KUKA KRL program: PPR-mid-01.src

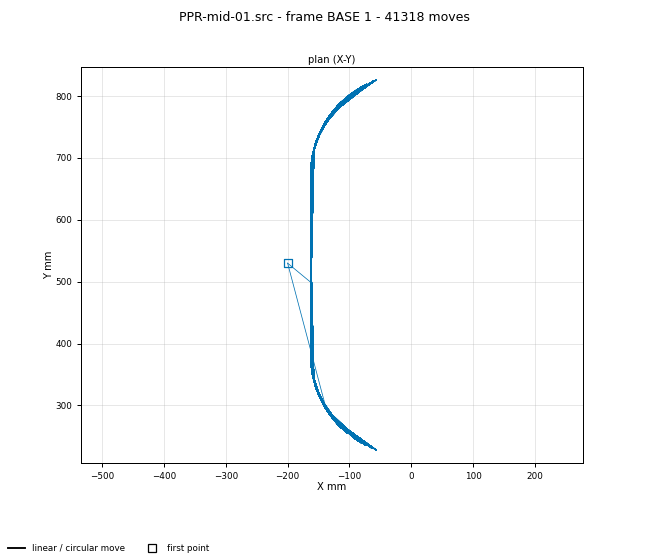
[picture p0: tool path of PPR-mid-01.src in frame BASE 1, 41318 of 41319 moves have a stored position in this frame; points joined in program order, loops and branches not executed]
&ACCESS RVEO
&REL 11
&PARAM TEMPLATE = C:\KRC\Roboter\Template\vorgabe
&PARAM EDITMASK = *
DEF variable_helical2( )
;FOLD INI
  ;FOLD BASISTECH INI
    GLOBAL INTERRUPT DECL 3 WHEN $STOPMESS==TRUE DO IR_STOPM ( )
    INTERRUPT ON 3
    BAS (#INITMOV,0 )
  ;ENDFOLD (BASISTECH INI)
 ;FOLD USER INI


    ;Make your modifications here
  ;ENDFOLD (USER INI)
;ENDFOLD (INI)
ACTION(#AXIS_RESET,34,1000,#NOERROR,ERROR_CODE)
;FOLD PTP HOME  Vel= 100 % DEFAULT;%{PE}%MKUKATPBASIS,%CMOVE,%VPTP,%P 1:PTP, 2:HOME, 3:, 5:100, 7:DEFAULT
$BWDSTART = FALSE
PDAT_ACT=PDEFAULT
FDAT_ACT=FHOME
BAS (#PTP_PARAMS,100 )
$H_POS=XHOME
PTP  XHOME
;ENDFOLD
BAS(#TOOL,1)
BAS(#BASE,1)
$VEL_AXIS[1]=100
$VEL_AXIS[2]=100
$VEL_AXIS[3]=100
$VEL_AXIS[4]=100
$VEL_AXIS[5]=100
$VEL_AXIS[6]=100
$VEL_EXTAX[1]=100
$VEL_EXTAX[2]=100

$ACC_AXIS[1]=100
$ACC_AXIS[2]=100
$ACC_AXIS[3]=100
$ACC_AXIS[4]=100
$ACC_AXIS[5]=100
$ACC_AXIS[6]=100
$ACC_EXTAX[1]=100
$ACC_EXTAX[2]=100

;;;;;;;;; postprocessing parameters (date 2024-01-25T18:14:56.965272)
; qxconst: -162.82
; qxconstarcys: -149.5,143.5
; qE3offset: 0.00
; qyoffset: 530.00
; qswitchsplit: 3
; qthinningtol: 0.2010
;;;;;;;;;

SLIN {X  -200.000, Y  +530.000, Z    +0.000, A    +0.000, E1    +0.000, E3    +0.000, E4    +0.000}

SLIN {X  -137.186, Y  +292.805, Z    +0.000, E1   +73.993, E3   +38.340}
HALT
SPLINE
SPL {X  -133.270, Y  +286.961, Z    +0.000, E1   +73.739, E3   +43.054}
SPL {X  -130.283, Y  +282.844, Z    +0.000, E1   +73.297, E3   +47.946}
SPL {X  -126.880, Y  +278.461, Z    +0.000, E1   +72.855, E3   +52.696}
SPL {X  -123.363, Y  +274.237, Z    +0.000, E1   +72.376, E3   +57.178}
SPL {X  -121.018, Y  +271.573, Z    +0.000, E1   +72.049, E3   +59.863}
SPL {X  -113.980, Y  +264.229, Z    +0.000, E1   +74.120, E3   +55.442}
SPL {X   -56.216, Y  +227.692, Z    +0.000, E1   +56.267, E3  +232.166}
ENDSPLINE

SPLINE
SPL {X  -126.995, Y  +278.604, Z    +0.000, E1   +59.937, E3  +404.406}
SPL {X  -150.196, Y  +317.640, Z    +0.000, E1   +49.956, E3  +412.861}
SPL {X  -157.261, Y  +338.316, Z    +0.000, E1   +40.017, E3  +414.556}
SPL {X  -160.924, Y  +355.726, Z    +0.000, E1   +27.715, E3  +414.997}
SPL {X  -162.423, Y  +369.141, Z    +0.000, E1   +15.207, E3  +415.432}
SPL {X  -162.811, Y  +378.755, Z    +0.000, E1    +4.616, E3  +415.347}
SPL {X  -162.820, Y  +382.684, Z    +0.000, E1    -0.227, E3  +414.902}
SPL {X  -162.820, Y  +385.721, Z    +0.000, E1    -8.371, E3  +414.717}
SPL {X  -162.820, Y  +388.532, Z    +0.000, E1   -16.412, E3  +414.604}
SPL {X  -162.820, Y  +392.558, Z    +0.000, E1   -27.778, E3  +414.692}
SPL {X  -162.820, Y  +400.474, Z    +0.000, E1   -46.251, E3  +414.556}
SPL {X  -162.820, Y  +414.510, Z    +0.000, E1   -65.115, E3  +413.999}
SPL {X  -162.820, Y  +465.064, Z    +0.000, E1   -76.269, E3  +423.847}
SPL {X  -157.184, Y  +715.968, Z    +0.000, E1   -76.600, E3  +519.805}
SPL {X  -156.461, Y  +718.560, Z    +0.000, E1   -75.553, E3  +533.225}
SPL {X  -151.911, Y  +732.096, Z    +0.000, E1   -75.235, E3  +543.779}
SPL {X  -146.569, Y  +744.407, Z    +0.000, E1   -74.677, E3  +555.583}
SPL {X  -142.375, Y  +752.491, Z    +0.000, E1   -74.335, E3  +562.610}
SPL {X  -139.539, Y  +757.399, Z    +0.000, E1   -73.892, E3  +568.808}
SPL {X  -136.017, Y  +762.997, Z    +0.000, E1   -73.579, E3  +573.990}
SPL {X  -133.089, Y  +767.296, Z    +0.000, E1   -73.251, E3  +578.448}
SPL {X  -129.985, Y  +771.553, Z    +0.000, E1   -72.801, E3  +583.442}
SPL {X  -126.581, Y  +775.909, Z    +0.000, E1   -72.426, E3  +587.753}
SPL {X  -122.528, Y  +780.725, Z    +0.000, E1   -71.905, E3  +592.773}
SPL {X  -116.189, Y  +787.563, Z    +0.000, E1   -72.978, E3  +592.058}
SPL {X   -57.587, Y  +825.796, Z    +0.000, E1   -56.753, E3  +747.309}
ENDSPLINE

SPLINE
SPL {X  -124.075, Y  +778.932, Z    +0.000, E1   -61.393, E3  +940.938}
SPL {X  -150.653, Y  +735.257, Z    +0.000, E1   -50.160, E3  +948.618}
SPL {X  -159.377, Y  +706.804, Z    +0.000, E1   -34.828, E3  +950.261}
SPL {X  -162.134, Y  +688.425, Z    +0.000, E1   -19.100, E3  +950.198}
SPL {X  -162.734, Y  +678.779, Z    +0.000, E1    -8.745, E3  +950.337}
SPL {X  -162.820, Y  +671.589, Z    +0.000, E1    -0.221, E3  +949.971}
SPL {X  -162.820, Y  +669.743, Z    +0.000, E1    +4.352, E3  +949.746}
SPL {X  -162.820, Y  +665.917, Z    +0.000, E1   +15.272, E3  +949.740}
SPL {X  -162.820, Y  +661.245, Z    +0.000, E1   +28.879, E3  +949.581}
SPL {X  -162.820, Y  +654.015, Z    +0.000, E1   +45.814, E3  +949.728}
SPL {X  -162.820, Y  +641.345, Z    +0.000, E1   +63.138, E3  +949.775}
SPL {X  -162.820, Y  +620.039, Z    +0.000, E1   +75.979, E3  +948.385}
SPL {X  -162.820, Y  +571.094, Z    +0.000, E1   +77.089, E3  +963.564}
SPL {X  -157.487, Y  +339.169, Z    +0.000, E1   +76.425, E3 +1056.668}
SPL {X  -156.386, Y  +335.181, Z    +0.000, E1   +75.555, E3 +1068.729}
SPL {X  -152.710, Y  +324.020, Z    +0.000, E1   +75.365, E3 +1076.539}
SPL {X  -139.497, Y  +296.529, Z    +0.000, E1   +77.231, E3 +1070.111}
ENDSPLINE

SPLINE
SPL {X  -139.792, Y  +297.022, Z    +0.000, E1   +76.273, E3 +1078.806}
ENDSPLINE

SPLINE
SPL {X  -138.933, Y  +295.600, Z    +0.000, E1   +75.173, E3 +1089.289}
SPL {X  -137.186, Y  +292.805, Z    +0.000, E1   +73.993, E3 +1099.879}
SPL {X  -133.270, Y  +286.961, Z    +0.000, E1   +73.739, E3 +1104.592}
SPL {X  -130.283, Y  +282.844, Z    +0.000, E1   +73.297, E3 +1109.484}
SPL {X  -127.795, Y  +279.610, Z    +0.000, E1   +72.860, E3 +1113.614}
SPL {X  -124.650, Y  +275.749, Z    +0.000, E1   +72.674, E3 +1116.533}
SPL {X  -121.687, Y  +272.322, Z    +0.000, E1   +72.100, E3 +1120.842}
SPL {X  -113.980, Y  +264.229, Z    +0.000, E1   +74.120, E3 +1116.980}
SPL {X   -56.216, Y  +227.692, Z    +0.000, E1   +56.267, E3 +1293.704}
ENDSPLINE

SPLINE
SPL {X  -126.995, Y  +278.604, Z    +0.000, E1   +59.937, E3 +1465.945}
SPL {X  -150.196, Y  +317.640, Z    +0.000, E1   +49.956, E3 +1474.400}
SPL {X  -157.261, Y  +338.316, Z    +0.000, E1   +40.017, E3 +1476.095}
SPL {X  -160.924, Y  +355.726, Z    +0.000, E1   +27.715, E3 +1476.535}
SPL {X  -162.423, Y  +369.141, Z    +0.000, E1   +15.207, E3 +1476.971}
SPL {X  -162.811, Y  +378.755, Z    +0.000, E1    +4.616, E3 +1476.885}
SPL {X  -162.820, Y  +382.684, Z    +0.000, E1    -0.227, E3 +1476.440}
SPL {X  -162.820, Y  +385.721, Z    +0.000, E1    -8.371, E3 +1476.256}
SPL {X  -162.820, Y  +388.532, Z    +0.000, E1   -16.412, E3 +1476.142}
SPL {X  -162.820, Y  +392.558, Z    +0.000, E1   -27.778, E3 +1476.231}
SPL {X  -162.820, Y  +398.468, Z    +0.000, E1   -42.446, E3 +1476.081}
SPL {X  -162.820, Y  +404.415, Z    +0.000, E1   -53.236, E3 +1476.121}
SPL {X  -162.820, Y  +414.510, Z    +0.000, E1   -65.115, E3 +1475.538}
SPL {X  -162.820, Y  +457.766, Z    +0.000, E1   -75.929, E3 +1483.374}
SPL {X  -162.820, Y  +471.144, Z    +0.000, E1   -76.496, E3 +1487.063}
SPL {X  -158.097, Y  +712.432, Z    +0.000, E1   -77.677, E3 +1567.773}
SPL {X  -156.557, Y  +718.224, Z    +0.000, E1   -75.715, E3 +1592.910}
SPL {X  -153.015, Y  +729.150, Z    +0.000, E1   -75.312, E3 +1602.852}
SPL {X  -149.053, Y  +739.025, Z    +0.000, E1   -74.952, E3 +1611.648}
SPL {X  -144.053, Y  +749.389, Z    +0.000, E1   -74.457, E3 +1621.639}
SPL {X  -139.539, Y  +757.399, Z    +0.000, E1   -73.892, E3 +1630.346}
SPL {X  -136.017, Y  +762.997, Z    +0.000, E1   -73.579, E3 +1635.529}
SPL {X  -133.089, Y  +767.296, Z    +0.000, E1   -73.251, E3 +1639.987}
SPL {X  -129.985, Y  +771.553, Z    +0.000, E1   -72.801, E3 +1644.981}
SPL {X  -126.581, Y  +775.909, Z    +0.000, E1   -72.426, E3 +1649.292}
SPL {X  -123.329, Y  +779.803, Z    +0.000, E1   -71.936, E3 +1653.674}
SPL {X  -119.291, Y  +784.315, Z    +0.000, E1   -72.148, E3 +1655.085}
SPL {X   -57.587, Y  +825.796, Z    +0.000, E1   -56.753, E3 +1808.848}
ENDSPLINE

SPLINE
SPL {X  -124.075, Y  +778.932, Z    +0.000, E1   -61.393, E3 +2002.477}
SPL {X  -150.653, Y  +735.257, Z    +0.000, E1   -50.160, E3 +2010.156}
SPL {X  -159.377, Y  +706.804, Z    +0.000, E1   -34.828, E3 +2011.800}
SPL {X  -162.134, Y  +688.425, Z    +0.000, E1   -19.100, E3 +2011.736}
SPL {X  -162.803, Y  +675.871, Z    +0.000, E1    -5.469, E3 +2011.920}
SPL {X  -162.820, Y  +671.500, Z    +0.000, E1    +0.000, E3 +2011.488}
SPL {X  -162.820, Y  +669.743, Z    +0.000, E1    +4.352, E3 +2011.284}
SPL {X  -162.820, Y  +665.917, Z    +0.000, E1   +15.272, E3 +2011.279}
SPL {X  -162.820, Y  +661.245, Z    +0.000, E1   +28.879, E3 +2011.120}
SPL {X  -162.820, Y  +654.015, Z    +0.000, E1   +45.814, E3 +2011.267}
SPL {X  -162.820, Y  +641.345, Z    +0.000, E1   +63.138, E3 +2011.314}
SPL {X  -162.820, Y  +620.039, Z    +0.000, E1   +75.979, E3 +2009.924}
SPL {X  -162.820, Y  +571.094, Z    +0.000, E1   +77.089, E3 +2025.102}
SPL {X  -157.487, Y  +339.169, Z    +0.000, E1   +76.425, E3 +2118.206}
SPL {X  -156.386, Y  +335.181, Z    +0.000, E1   +75.555, E3 +2130.267}
SPL {X  -152.710, Y  +324.020, Z    +0.000, E1   +75.365, E3 +2138.077}
SPL {X  -139.497, Y  +296.529, Z    +0.000, E1   +77.231, E3 +2131.649}
ENDSPLINE

SPLINE
SPL {X  -139.792, Y  +297.022, Z    +0.000, E1   +76.273, E3 +2140.344}
ENDSPLINE

SPLINE
SPL {X  -138.933, Y  +295.600, Z    +0.000, E1   +75.173, E3 +2150.827}
SPL {X  -137.186, Y  +292.805, Z    +0.000, E1   +73.993, E3 +2161.417}
SPL {X  -133.270, Y  +286.961, Z    +0.000, E1   +73.739, E3 +2166.131}
SPL {X  -130.283, Y  +282.844, Z    +0.000, E1   +73.297, E3 +2171.023}
SPL {X  -127.795, Y  +279.610, Z    +0.000, E1   +72.860, E3 +2175.153}
SPL {X  -124.650, Y  +275.749, Z    +0.000, E1   +72.674, E3 +2178.071}
SPL {X  -121.687, Y  +272.322, Z    +0.000, E1   +72.100, E3 +2182.381}
SPL {X  -113.980, Y  +264.229, Z    +0.000, E1   +74.120, E3 +2178.519}
SPL {X   -56.216, Y  +227.692, Z    +0.000, E1   +56.267, E3 +2355.243}
ENDSPLINE

SPLINE
SPL {X  -126.995, Y  +278.604, Z    +0.000, E1   +59.937, E3 +2527.483}
SPL {X  -150.196, Y  +317.640, Z    +0.000, E1   +49.956, E3 +2535.938}
SPL {X  -157.261, Y  +338.316, Z    +0.000, E1   +40.017, E3 +2537.633}
SPL {X  -160.924, Y  +355.726, Z    +0.000, E1   +27.715, E3 +2538.074}
SPL {X  -162.423, Y  +369.141, Z    +0.000, E1   +15.207, E3 +2538.509}
SPL {X  -162.811, Y  +378.755, Z    +0.000, E1    +4.616, E3 +2538.424}
SPL {X  -162.820, Y  +382.684, Z    +0.000, E1    -0.227, E3 +2537.978}
SPL {X  -162.820, Y  +387.227, Z    +0.000, E1   -12.320, E3 +2537.733}
SPL {X  -162.820, Y  +392.558, Z    +0.000, E1   -27.778, E3 +2537.769}
SPL {X  -162.820, Y  +400.474, Z    +0.000, E1   -46.251, E3 +2537.633}
SPL {X  -162.820, Y  +414.510, Z    +0.000, E1   -65.115, E3 +2537.076}
SPL {X  -162.820, Y  +465.064, Z    +0.000, E1   -76.269, E3 +2546.924}
SPL {X  -158.097, Y  +712.432, Z    +0.000, E1   -77.677, E3 +2629.312}
SPL {X  -156.557, Y  +718.224, Z    +0.000, E1   -75.715, E3 +2654.448}
SPL {X  -151.911, Y  +732.096, Z    +0.000, E1   -75.235, E3 +2666.856}
SPL {X  -146.569, Y  +744.407, Z    +0.000, E1   -74.677, E3 +2678.660}
SPL {X  -142.375, Y  +752.491, Z    +0.000, E1   -74.335, E3 +2685.687}
SPL {X  -139.539, Y  +757.399, Z    +0.000, E1   -73.892, E3 +2691.885}
SPL {X  -136.017, Y  +762.997, Z    +0.000, E1   -73.579, E3 +2697.067}
SPL {X  -133.089, Y  +767.296, Z    +0.000, E1   -73.251, E3 +2701.525}
SPL {X  -129.985, Y  +771.553, Z    +0.000, E1   -72.801, E3 +2706.519}
SPL {X  -126.581, Y  +775.909, Z    +0.000, E1   -72.426, E3 +2710.830}
SPL {X  -123.329, Y  +779.803, Z    +0.000, E1   -71.936, E3 +2715.212}
SPL {X  -119.291, Y  +784.315, Z    +0.000, E1   -72.148, E3 +2716.624}
SPL {X   -57.587, Y  +825.796, Z    +0.000, E1   -56.753, E3 +2870.386}
ENDSPLINE

SPLINE
SPL {X  -124.075, Y  +778.932, Z    +0.000, E1   -61.393, E3 +3064.015}
SPL {X  -150.653, Y  +735.257, Z    +0.000, E1   -50.160, E3 +3071.695}
SPL {X  -159.377, Y  +706.804, Z    +0.000, E1   -34.828, E3 +3073.338}
SPL {X  -162.134, Y  +688.425, Z    +0.000, E1   -19.100, E3 +3073.275}
SPL {X  -162.803, Y  +675.871, Z    +0.000, E1    -5.469, E3 +3073.459}
SPL {X  -162.820, Y  +671.500, Z    +0.000, E1    +0.000, E3 +3073.027}
SPL {X  -162.820, Y  +669.743, Z    +0.000, E1    +4.352, E3 +3072.822}
SPL {X  -162.820, Y  +665.917, Z    +0.000, E1   +15.272, E3 +3072.817}
SPL {X  -162.820, Y  +661.245, Z    +0.000, E1   +28.879, E3 +3072.658}
SPL {X  -162.820, Y  +654.015, Z    +0.000, E1   +45.814, E3 +3072.805}
SPL {X  -162.820, Y  +641.345, Z    +0.000, E1   +63.138, E3 +3072.852}
SPL {X  -162.820, Y  +620.039, Z    +0.000, E1   +75.979, E3 +3071.462}
SPL {X  -162.820, Y  +571.094, Z    +0.000, E1   +77.089, E3 +3086.641}
SPL {X  -157.487, Y  +339.169, Z    +0.000, E1   +76.425, E3 +3179.745}
SPL {X  -156.386, Y  +335.181, Z    +0.000, E1   +75.555, E3 +3191.805}
SPL {X  -152.710, Y  +324.020, Z    +0.000, E1   +75.365, E3 +3199.616}
SPL {X  -139.497, Y  +296.529, Z    +0.000, E1   +77.231, E3 +3193.188}
ENDSPLINE

SPLINE
SPL {X  -139.792, Y  +297.022, Z    +0.000, E1   +76.273, E3 +3201.883}
ENDSPLINE

SPLINE
SPL {X  -138.933, Y  +295.600, Z    +0.000, E1   +75.173, E3 +3212.365}
SPL {X  -137.186, Y  +292.805, Z    +0.000, E1   +73.993, E3 +3222.956}
SPL {X  -133.270, Y  +286.961, Z    +0.000, E1   +73.739, E3 +3227.669}
SPL {X  -130.283, Y  +282.844, Z    +0.000, E1   +73.297, E3 +3232.561}
SPL {X  -127.795, Y  +279.610, Z    +0.000, E1   +72.860, E3 +3236.691}
SPL {X  -124.650, Y  +275.749, Z    +0.000, E1   +72.674, E3 +3239.610}
SPL {X  -121.687, Y  +272.322, Z    +0.000, E1   +72.100, E3 +3243.919}
SPL {X  -113.980, Y  +264.229, Z    +0.000, E1   +74.120, E3 +3240.057}
SPL {X   -56.216, Y  +227.692, Z    +0.000, E1   +56.267, E3 +3416.781}
ENDSPLINE

SPLINE
SPL {X  -126.995, Y  +278.604, Z    +0.000, E1   +59.937, E3 +3589.021}
SPL {X  -150.196, Y  +317.640, Z    +0.000, E1   +49.956, E3 +3597.477}
SPL {X  -157.261, Y  +338.316, Z    +0.000, E1   +40.017, E3 +3599.172}
SPL {X  -160.924, Y  +355.726, Z    +0.000, E1   +27.715, E3 +3599.612}
SPL {X  -162.423, Y  +369.141, Z    +0.000, E1   +15.207, E3 +3600.048}
SPL {X  -162.811, Y  +378.755, Z    +0.000, E1    +4.616, E3 +3599.962}
SPL {X  -162.820, Y  +382.684, Z    +0.000, E1    -0.227, E3 +3599.517}
SPL {X  -162.820, Y  +387.227, Z    +0.000, E1   -12.320, E3 +3599.272}
SPL {X  -162.820, Y  +392.558, Z    +0.000, E1   -27.778, E3 +3599.308}
SPL {X  -162.820, Y  +400.474, Z    +0.000, E1   -46.251, E3 +3599.172}
SPL {X  -162.820, Y  +414.510, Z    +0.000, E1   -65.115, E3 +3598.615}
SPL {X  -162.820, Y  +465.064, Z    +0.000, E1   -76.269, E3 +3608.463}
SPL {X  -158.097, Y  +712.432, Z    +0.000, E1   -77.677, E3 +3690.850}
SPL {X  -156.557, Y  +718.224, Z    +0.000, E1   -75.715, E3 +3715.987}
SPL {X  -151.911, Y  +732.096, Z    +0.000, E1   -75.235, E3 +3728.394}
SPL {X  -146.569, Y  +744.407, Z    +0.000, E1   -74.677, E3 +3740.198}
SPL {X  -142.375, Y  +752.491, Z    +0.000, E1   -74.335, E3 +3747.226}
SPL {X  -139.539, Y  +757.399, Z    +0.000, E1   -73.892, E3 +3753.423}
SPL {X  -136.017, Y  +762.997, Z    +0.000, E1   -73.579, E3 +3758.606}
SPL {X  -133.089, Y  +767.296, Z    +0.000, E1   -73.251, E3 +3763.064}
SPL {X  -129.985, Y  +771.553, Z    +0.000, E1   -72.801, E3 +3768.057}
SPL {X  -126.581, Y  +775.909, Z    +0.000, E1   -72.426, E3 +3772.369}
SPL {X  -123.329, Y  +779.803, Z    +0.000, E1   -71.936, E3 +3776.750}
SPL {X  -119.291, Y  +784.315, Z    +0.000, E1   -72.148, E3 +3778.162}
SPL {X   -57.587, Y  +825.796, Z    +0.000, E1   -56.753, E3 +3931.925}
ENDSPLINE

SPLINE
SPL {X  -124.075, Y  +778.932, Z    +0.000, E1   -61.393, E3 +4125.554}
SPL {X  -150.653, Y  +735.257, Z    +0.000, E1   -50.160, E3 +4133.233}
SPL {X  -159.377, Y  +706.804, Z    +0.000, E1   -34.828, E3 +4134.876}
SPL {X  -162.134, Y  +688.425, Z    +0.000, E1   -19.100, E3 +4134.813}
SPL {X  -162.803, Y  +675.871, Z    +0.000, E1    -5.469, E3 +4134.997}
SPL {X  -162.820, Y  +671.500, Z    +0.000, E1    +0.000, E3 +4134.565}
SPL {X  -162.820, Y  +669.743, Z    +0.000, E1    +4.352, E3 +4134.361}
SPL {X  -162.820, Y  +665.917, Z    +0.000, E1   +15.272, E3 +4134.355}
SPL {X  -162.820, Y  +661.245, Z    +0.000, E1   +28.879, E3 +4134.197}
SPL {X  -162.820, Y  +654.015, Z    +0.000, E1   +45.814, E3 +4134.344}
SPL {X  -162.820, Y  +641.345, Z    +0.000, E1   +63.138, E3 +4134.391}
SPL {X  -162.820, Y  +620.039, Z    +0.000, E1   +75.979, E3 +4133.001}
SPL {X  -162.820, Y  +571.094, Z    +0.000, E1   +77.089, E3 +4148.179}
SPL {X  -157.487, Y  +339.169, Z    +0.000, E1   +76.425, E3 +4241.283}
SPL {X  -156.386, Y  +335.181, Z    +0.000, E1   +75.555, E3 +4253.344}
SPL {X  -152.710, Y  +324.020, Z    +0.000, E1   +75.365, E3 +4261.154}
SPL {X  -139.497, Y  +296.529, Z    +0.000, E1   +77.231, E3 +4254.726}
ENDSPLINE

SPLINE
SPL {X  -139.792, Y  +297.022, Z    +0.000, E1   +76.273, E3 +4263.421}
ENDSPLINE

SPLINE
SPL {X  -138.933, Y  +295.600, Z    +0.000, E1   +75.173, E3 +4273.904}
SPL {X  -137.186, Y  +292.805, Z    +0.000, E1   +73.993, E3 +4284.494}
SPL {X  -133.270, Y  +286.961, Z    +0.000, E1   +73.739, E3 +4289.208}
SPL {X  -130.283, Y  +282.844, Z    +0.000, E1   +73.297, E3 +4294.100}
SPL {X  -127.795, Y  +279.610, Z    +0.000, E1   +72.860, E3 +4298.230}
SPL {X  -124.650, Y  +275.749, Z    +0.000, E1   +72.674, E3 +4301.148}
SPL {X  -121.687, Y  +272.322, Z    +0.000, E1   +72.100, E3 +4305.457}
SPL {X  -113.980, Y  +264.229, Z    +0.000, E1   +74.120, E3 +4301.596}
SPL {X   -56.216, Y  +227.692, Z    +0.000, E1   +56.267, E3 +4478.320}
ENDSPLINE

SPLINE
SPL {X  -126.995, Y  +278.604, Z    +0.000, E1   +59.937, E3 +4650.560}
SPL {X  -150.196, Y  +317.640, Z    +0.000, E1   +49.956, E3 +4659.015}
SPL {X  -157.261, Y  +338.316, Z    +0.000, E1   +40.017, E3 +4660.710}
SPL {X  -160.924, Y  +355.726, Z    +0.000, E1   +27.715, E3 +4661.151}
SPL {X  -162.423, Y  +369.141, Z    +0.000, E1   +15.207, E3 +4661.586}
SPL {X  -162.811, Y  +378.755, Z    +0.000, E1    +4.616, E3 +4661.501}
SPL {X  -162.820, Y  +382.684, Z    +0.000, E1    -0.227, E3 +4661.055}
SPL {X  -162.820, Y  +387.227, Z    +0.000, E1   -12.320, E3 +4660.810}
SPL {X  -162.820, Y  +392.558, Z    +0.000, E1   -27.778, E3 +4660.846}
SPL {X  -162.820, Y  +400.474, Z    +0.000, E1   -46.251, E3 +4660.710}
SPL {X  -162.820, Y  +414.510, Z    +0.000, E1   -65.115, E3 +4660.153}
SPL {X  -162.820, Y  +465.064, Z    +0.000, E1   -76.269, E3 +4670.001}
SPL {X  -158.097, Y  +712.432, Z    +0.000, E1   -77.677, E3 +4752.389}
SPL {X  -156.557, Y  +718.224, Z    +0.000, E1   -75.715, E3 +4777.525}
SPL {X  -151.911, Y  +732.096, Z    +0.000, E1   -75.235, E3 +4789.932}
SPL {X  -146.569, Y  +744.407, Z    +0.000, E1   -74.677, E3 +4801.737}
SPL {X  -142.375, Y  +752.491, Z    +0.000, E1   -74.335, E3 +4808.764}
SPL {X  -139.539, Y  +757.399, Z    +0.000, E1   -73.892, E3 +4814.962}
SPL {X  -136.017, Y  +762.997, Z    +0.000, E1   -73.579, E3 +4820.144}
SPL {X  -133.089, Y  +767.296, Z    +0.000, E1   -73.251, E3 +4824.602}
SPL {X  -129.985, Y  +771.553, Z    +0.000, E1   -72.801, E3 +4829.596}
SPL {X  -126.581, Y  +775.909, Z    +0.000, E1   -72.426, E3 +4833.907}
SPL {X  -123.329, Y  +779.803, Z    +0.000, E1   -71.936, E3 +4838.289}
SPL {X  -119.291, Y  +784.315, Z    +0.000, E1   -72.148, E3 +4839.701}
SPL {X   -57.587, Y  +825.796, Z    +0.000, E1   -56.753, E3 +4993.463}
ENDSPLINE

SPLINE
SPL {X  -124.075, Y  +778.932, Z    +0.000, E1   -61.393, E3 +5187.092}
SPL {X  -150.653, Y  +735.257, Z    +0.000, E1   -50.160, E3 +5194.772}
SPL {X  -159.377, Y  +706.804, Z    +0.000, E1   -34.828, E3 +5196.415}
SPL {X  -162.134, Y  +688.425, Z    +0.000, E1   -19.100, E3 +5196.352}
SPL {X  -162.803, Y  +675.871, Z    +0.000, E1    -5.469, E3 +5196.536}
SPL {X  -162.820, Y  +671.500, Z    +0.000, E1    +0.000, E3 +5196.104}
SPL {X  -162.820, Y  +669.743, Z    +0.000, E1    +4.352, E3 +5195.899}
SPL {X  -162.820, Y  +665.917, Z    +0.000, E1   +15.272, E3 +5195.894}
SPL {X  -162.820, Y  +661.245, Z    +0.000, E1   +28.879, E3 +5195.735}
SPL {X  -162.820, Y  +654.015, Z    +0.000, E1   +45.814, E3 +5195.882}
SPL {X  -162.820, Y  +641.345, Z    +0.000, E1   +63.138, E3 +5195.929}
SPL {X  -162.820, Y  +620.039, Z    +0.000, E1   +75.979, E3 +5194.539}
SPL {X  -162.820, Y  +571.094, Z    +0.000, E1   +77.089, E3 +5209.718}
SPL {X  -157.487, Y  +339.169, Z    +0.000, E1   +76.425, E3 +5302.822}
SPL {X  -156.386, Y  +335.181, Z    +0.000, E1   +75.555, E3 +5314.882}
SPL {X  -152.710, Y  +324.020, Z    +0.000, E1   +75.365, E3 +5322.693}
SPL {X  -139.497, Y  +296.529, Z    +0.000, E1   +77.231, E3 +5316.264}
ENDSPLINE

SPLINE
SPL {X  -139.520, Y  +296.568, Z    +0.000, E1   +75.884, E3 +5328.912}
ENDSPLINE

SPLINE
SPL {X  -138.554, Y  +294.984, Z    +0.000, E1   +74.772, E3 +5338.793}
SPL {X  -137.186, Y  +292.805, Z    +0.000, E1   +73.993, E3 +5346.033}
SPL {X  -133.270, Y  +286.961, Z    +0.000, E1   +73.739, E3 +5350.746}
SPL {X  -130.283, Y  +282.844, Z    +0.000, E1   +73.297, E3 +5355.638}
SPL {X  -126.880, Y  +278.461, Z    +0.000, E1   +72.855, E3 +5360.389}
SPL {X  -123.363, Y  +274.237, Z    +0.000, E1   +72.376, E3 +5364.871}
SPL {X  -121.018, Y  +271.573, Z    +0.000, E1   +72.049, E3 +5367.556}
SPL {X  -113.980, Y  +264.229, Z    +0.000, E1   +74.120, E3 +5363.134}
SPL {X   -56.216, Y  +227.692, Z    +0.000, E1   +56.267, E3 +5539.858}
ENDSPLINE

SPLINE
SPL {X  -126.995, Y  +278.604, Z    +0.000, E1   +59.937, E3 +5712.098}
SPL {X  -150.196, Y  +317.640, Z    +0.000, E1   +49.956, E3 +5720.553}
SPL {X  -157.261, Y  +338.316, Z    +0.000, E1   +40.017, E3 +5722.249}
SPL {X  -160.924, Y  +355.726, Z    +0.000, E1   +27.715, E3 +5722.689}
SPL {X  -162.423, Y  +369.141, Z    +0.000, E1   +15.207, E3 +5723.125}
SPL {X  -162.811, Y  +378.755, Z    +0.000, E1    +4.616, E3 +5723.039}
SPL {X  -162.820, Y  +382.684, Z    +0.000, E1    -0.227, E3 +5722.594}
SPL {X  -162.820, Y  +385.721, Z    +0.000, E1    -8.371, E3 +5722.409}
SPL {X  -162.820, Y  +388.532, Z    +0.000, E1   -16.412, E3 +5722.296}
SPL {X  -162.820, Y  +392.558, Z    +0.000, E1   -27.778, E3 +5722.385}
SPL {X  -162.820, Y  +400.474, Z    +0.000, E1   -46.251, E3 +5722.248}
SPL {X  -162.820, Y  +414.510, Z    +0.000, E1   -65.115, E3 +5721.692}
SPL {X  -162.820, Y  +465.064, Z    +0.000, E1   -76.269, E3 +5731.540}
SPL {X  -157.184, Y  +715.968, Z    +0.000, E1   -76.600, E3 +5827.497}
SPL {X  -156.461, Y  +718.560, Z    +0.000, E1   -75.553, E3 +5840.917}
SPL {X  -153.015, Y  +729.150, Z    +0.000, E1   -75.312, E3 +5849.006}
SPL {X  -149.053, Y  +739.025, Z    +0.000, E1   -74.952, E3 +5857.802}
SPL {X  -144.053, Y  +749.389, Z    +0.000, E1   -74.457, E3 +5867.793}
SPL {X  -139.539, Y  +757.399, Z    +0.000, E1   -73.892, E3 +5876.500}
SPL {X  -136.017, Y  +762.997, Z    +0.000, E1   -73.579, E3 +5881.683}
SPL {X  -133.089, Y  +767.296, Z    +0.000, E1   -73.251, E3 +5886.141}
SPL {X  -129.985, Y  +771.553, Z    +0.000, E1   -72.801, E3 +5891.134}
SPL {X  -126.581, Y  +775.909, Z    +0.000, E1   -72.426, E3 +5895.446}
SPL {X  -123.329, Y  +779.803, Z    +0.000, E1   -71.936, E3 +5899.827}
SPL {X  -119.291, Y  +784.315, Z    +0.000, E1   -72.148, E3 +5901.239}
SPL {X   -57.587, Y  +825.796, Z    +0.000, E1   -56.753, E3 +6055.002}
ENDSPLINE

SPLINE
SPL {X  -124.075, Y  +778.932, Z    +0.000, E1   -61.393, E3 +6248.631}
SPL {X  -147.028, Y  +743.450, Z    +0.000, E1   -53.078, E3 +6255.368}
SPL {X  -152.552, Y  +730.406, Z    +0.000, E1   -48.136, E3 +6256.786}
SPL {X  -159.377, Y  +706.804, Z    +0.000, E1   -34.828, E3 +6257.953}
SPL {X  -162.134, Y  +688.425, Z    +0.000, E1   -19.100, E3 +6257.890}
SPL {X  -162.803, Y  +675.871, Z    +0.000, E1    -5.469, E3 +6258.074}
SPL {X  -162.820, Y  +671.500, Z    +0.000, E1    +0.000, E3 +6257.642}
SPL {X  -162.820, Y  +669.743, Z    +0.000, E1    +4.352, E3 +6257.438}
SPL {X  -162.820, Y  +665.917, Z    +0.000, E1   +15.272, E3 +6257.432}
SPL {X  -162.820, Y  +659.880, Z    +0.000, E1   +32.256, E3 +6257.344}
SPL {X  -162.820, Y  +652.069, Z    +0.000, E1   +49.663, E3 +6257.369}
SPL {X  -162.820, Y  +641.345, Z    +0.000, E1   +63.138, E3 +6257.468}
SPL {X  -162.820, Y  +620.039, Z    +0.000, E1   +75.979, E3 +6256.078}
SPL {X  -162.820, Y  +578.479, Z    +0.000, E1   +77.260, E3 +6268.348}
SPL {X  -162.820, Y  +557.052, Z    +0.000, E1   +76.772, E3 +6276.829}
SPL {X  -157.487, Y  +339.169, Z    +0.000, E1   +76.425, E3 +6364.360}
SPL {X  -156.386, Y  +335.181, Z    +0.000, E1   +75.555, E3 +6376.421}
SPL {X  -152.710, Y  +324.020, Z    +0.000, E1   +75.365, E3 +6384.231}
SPL {X  -139.497, Y  +296.529, Z    +0.000, E1   +77.231, E3 +6377.803}
ENDSPLINE

SPLINE
SPL {X  -139.520, Y  +296.568, Z    +0.000, E1   +75.884, E3 +6390.450}
ENDSPLINE

SPLINE
SPL {X  -138.554, Y  +294.984, Z    +0.000, E1   +74.772, E3 +6400.331}
SPL {X  -137.186, Y  +292.805, Z    +0.000, E1   +73.993, E3 +6407.571}
SPL {X  -133.270, Y  +286.961, Z    +0.000, E1   +73.739, E3 +6412.285}
SPL {X  -130.283, Y  +282.844, Z    +0.000, E1   +73.297, E3 +6417.177}
SPL {X  -126.880, Y  +278.461, Z    +0.000, E1   +72.855, E3 +6421.927}
SPL {X  -123.363, Y  +274.237, Z    +0.000, E1   +72.376, E3 +6426.409}
SPL {X  -121.018, Y  +271.573, Z    +0.000, E1   +72.049, E3 +6429.094}
SPL {X  -113.980, Y  +264.229, Z    +0.000, E1   +74.120, E3 +6424.673}
SPL {X   -56.216, Y  +227.692, Z    +0.000, E1   +56.267, E3 +6601.397}
ENDSPLINE

SPLINE
SPL {X  -126.995, Y  +278.604, Z    +0.000, E1   +59.937, E3 +6773.637}
SPL {X  -150.196, Y  +317.640, Z    +0.000, E1   +49.956, E3 +6782.092}
SPL {X  -157.261, Y  +338.316, Z    +0.000, E1   +40.017, E3 +6783.787}
SPL {X  -160.924, Y  +355.726, Z    +0.000, E1   +27.715, E3 +6784.228}
SPL {X  -162.423, Y  +369.141, Z    +0.000, E1   +15.207, E3 +6784.663}
SPL {X  -162.811, Y  +378.755, Z    +0.000, E1    +4.616, E3 +6784.578}
SPL {X  -162.820, Y  +382.684, Z    +0.000, E1    -0.227, E3 +6784.132}
SPL {X  -162.820, Y  +385.721, Z    +0.000, E1    -8.371, E3 +6783.948}
SPL {X  -162.820, Y  +388.532, Z    +0.000, E1   -16.412, E3 +6783.834}
SPL {X  -162.820, Y  +392.558, Z    +0.000, E1   -27.778, E3 +6783.923}
SPL {X  -162.820, Y  +398.468, Z    +0.000, E1   -42.446, E3 +6783.774}
SPL {X  -162.820, Y  +404.415, Z    +0.000, E1   -53.236, E3 +6783.813}
SPL {X  -162.820, Y  +414.510, Z    +0.000, E1   -65.115, E3 +6783.230}
SPL {X  -162.820, Y  +457.766, Z    +0.000, E1   -75.929, E3 +6791.066}
SPL {X  -162.820, Y  +471.144, Z    +0.000, E1   -76.496, E3 +6794.755}
SPL {X  -158.097, Y  +712.432, Z    +0.000, E1   -77.677, E3 +6875.466}
SPL {X  -156.557, Y  +718.224, Z    +0.000, E1   -75.715, E3 +6900.602}
SPL {X  -151.911, Y  +732.096, Z    +0.000, E1   -75.235, E3 +6913.009}
SPL {X  -146.569, Y  +744.407, Z    +0.000, E1   -74.677, E3 +6924.814}
SPL {X  -142.375, Y  +752.491, Z    +0.000, E1   -74.335, E3 +6931.841}
SPL {X  -139.539, Y  +757.399, Z    +0.000, E1   -73.892, E3 +6938.039}
SPL {X  -136.017, Y  +762.997, Z    +0.000, E1   -73.579, E3 +6943.221}
SPL {X  -133.089, Y  +767.296, Z    +0.000, E1   -73.251, E3 +6947.679}
SPL {X  -129.985, Y  +771.553, Z    +0.000, E1   -72.801, E3 +6952.673}
SPL {X  -126.581, Y  +775.909, Z    +0.000, E1   -72.426, E3 +6956.984}
SPL {X  -123.329, Y  +779.803, Z    +0.000, E1   -71.936, E3 +6961.366}
SPL {X  -119.291, Y  +784.315, Z    +0.000, E1   -72.148, E3 +6962.778}
SPL {X   -57.587, Y  +825.796, Z    +0.000, E1   -56.753, E3 +7116.540}
ENDSPLINE

SPLINE
SPL {X  -124.075, Y  +778.932, Z    +0.000, E1   -61.393, E3 +7310.169}
SPL {X  -150.653, Y  +735.257, Z    +0.000, E1   -50.160, E3 +7317.848}
SPL {X  -159.377, Y  +706.804, Z    +0.000, E1   -34.828, E3 +7319.492}
SPL {X  -162.134, Y  +688.425, Z    +0.000, E1   -19.100, E3 +7319.429}
SPL {X  -162.734, Y  +678.779, Z    +0.000, E1    -8.745, E3 +7319.568}
SPL {X  -162.820, Y  +671.589, Z    +0.000, E1    -0.221, E3 +7319.202}
SPL {X  -162.820, Y  +669.743, Z    +0.000, E1    +4.352, E3 +7318.976}
SPL {X  -162.820, Y  +665.917, Z    +0.000, E1   +15.272, E3 +7318.971}
SPL {X  -162.820, Y  +659.880, Z    +0.000, E1   +32.256, E3 +7318.882}
SPL {X  -162.820, Y  +652.069, Z    +0.000, E1   +49.663, E3 +7318.908}
SPL {X  -162.820, Y  +641.345, Z    +0.000, E1   +63.138, E3 +7319.006}
SPL {X  -162.820, Y  +620.039, Z    +0.000, E1   +75.979, E3 +7317.616}
SPL {X  -162.820, Y  +571.094, Z    +0.000, E1   +77.089, E3 +7332.795}
SPL {X  -158.110, Y  +341.619, Z    +0.000, E1   +77.339, E3 +7414.444}
SPL {X  -156.597, Y  +335.917, Z    +0.000, E1   +75.680, E3 +7436.288}
SPL {X  -152.710, Y  +324.020, Z    +0.000, E1   +75.365, E3 +7445.770}
SPL {X  -139.497, Y  +296.529, Z    +0.000, E1   +77.231, E3 +7439.341}
ENDSPLINE

SPLINE
SPL {X  -139.792, Y  +297.022, Z    +0.000, E1   +76.273, E3 +7448.037}
ENDSPLINE

SPLINE
SPL {X  -138.933, Y  +295.600, Z    +0.000, E1   +75.173, E3 +7458.519}
SPL {X  -137.186, Y  +292.805, Z    +0.000, E1   +73.993, E3 +7469.110}
SPL {X  -133.270, Y  +286.961, Z    +0.000, E1   +73.739, E3 +7473.823}
SPL {X  -130.283, Y  +282.844, Z    +0.000, E1   +73.297, E3 +7478.715}
SPL {X  -126.880, Y  +278.461, Z    +0.000, E1   +72.855, E3 +7483.466}
SPL {X  -123.363, Y  +274.237, Z    +0.000, E1   +72.376, E3 +7487.948}
SPL {X  -121.018, Y  +271.573, Z    +0.000, E1   +72.049, E3 +7490.633}
SPL {X  -113.980, Y  +264.229, Z    +0.000, E1   +74.120, E3 +7486.211}
SPL {X   -56.216, Y  +227.692, Z    +0.000, E1   +56.267, E3 +7662.935}
ENDSPLINE

SPLINE
SPL {X  -126.995, Y  +278.604, Z    +0.000, E1   +59.937, E3 +7835.175}
SPL {X  -150.196, Y  +317.640, Z    +0.000, E1   +49.956, E3 +7843.630}
SPL {X  -157.261, Y  +338.316, Z    +0.000, E1   +40.017, E3 +7845.326}
SPL {X  -160.924, Y  +355.726, Z    +0.000, E1   +27.715, E3 +7845.766}
SPL {X  -162.423, Y  +369.141, Z    +0.000, E1   +15.207, E3 +7846.202}
SPL {X  -162.811, Y  +378.755, Z    +0.000, E1    +4.616, E3 +7846.116}
SPL {X  -162.820, Y  +382.684, Z    +0.000, E1    -0.227, E3 +7845.671}
SPL {X  -162.820, Y  +385.721, Z    +0.000, E1    -8.371, E3 +7845.486}
SPL {X  -162.820, Y  +388.532, Z    +0.000, E1   -16.412, E3 +7845.373}
SPL {X  -162.820, Y  +392.558, Z    +0.000, E1   -27.778, E3 +7845.462}
SPL {X  -162.820, Y  +400.474, Z    +0.000, E1   -46.251, E3 +7845.325}
SPL {X  -162.820, Y  +414.510, Z    +0.000, E1   -65.115, E3 +7844.769}
SPL {X  -162.820, Y  +465.064, Z    +0.000, E1   -76.269, E3 +7854.617}
SPL {X  -157.184, Y  +715.968, Z    +0.000, E1   -76.600, E3 +7950.574}
SPL {X  -156.461, Y  +718.560, Z    +0.000, E1   -75.553, E3 +7963.994}
SPL {X  -151.911, Y  +732.096, Z    +0.000, E1   -75.235, E3 +7974.548}
SPL {X  -146.569, Y  +744.407, Z    +0.000, E1   -74.677, E3 +7986.352}
SPL {X  -142.375, Y  +752.491, Z    +0.000, E1   -74.335, E3 +7993.379}
SPL {X  -139.539, Y  +757.399, Z    +0.000, E1   -73.892, E3 +7999.577}
SPL {X  -136.017, Y  +762.997, Z    +0.000, E1   -73.579, E3 +8004.759}
SPL {X  -133.089, Y  +767.296, Z    +0.000, E1   -73.251, E3 +8009.218}
SPL {X  -129.985, Y  +771.553, Z    +0.000, E1   -72.801, E3 +8014.211}
SPL {X  -126.581, Y  +775.909, Z    +0.000, E1   -72.426, E3 +8018.522}
SPL {X  -122.528, Y  +780.725, Z    +0.000, E1   -71.905, E3 +8023.542}
SPL {X  -116.189, Y  +787.563, Z    +0.000, E1   -72.978, E3 +8022.827}
SPL {X   -57.587, Y  +825.796, Z    +0.000, E1   -56.753, E3 +8178.079}
ENDSPLINE

SPLINE
SPL {X  -124.075, Y  +778.932, Z    +0.000, E1   -61.393, E3 +8371.708}
SPL {X  -150.653, Y  +735.257, Z    +0.000, E1   -50.160, E3 +8379.387}
SPL {X  -159.377, Y  +706.804, Z    +0.000, E1   -34.828, E3 +8381.030}
SPL {X  -162.134, Y  +688.425, Z    +0.000, E1   -19.100, E3 +8380.967}
SPL {X  -162.734, Y  +678.779, Z    +0.000, E1    -8.745, E3 +8381.106}
SPL {X  -162.820, Y  +671.589, Z    +0.000, E1    -0.221, E3 +8380.741}
SPL {X  -162.820, Y  +669.743, Z    +0.000, E1    +4.352, E3 +8380.515}
SPL {X  -162.820, Y  +665.917, Z    +0.000, E1   +15.272, E3 +8380.509}
SPL {X  -162.820, Y  +661.245, Z    +0.000, E1   +28.879, E3 +8380.350}
SPL {X  -162.820, Y  +654.015, Z    +0.000, E1   +45.814, E3 +8380.498}
SPL {X  -162.820, Y  +641.345, Z    +0.000, E1   +63.138, E3 +8380.545}
SPL {X  -162.820, Y  +620.039, Z    +0.000, E1   +75.979, E3 +8379.154}
SPL {X  -162.820, Y  +571.094, Z    +0.000, E1   +77.089, E3 +8394.333}
SPL {X  -158.110, Y  +341.619, Z    +0.000, E1   +77.339, E3 +8475.983}
SPL {X  -156.597, Y  +335.917, Z    +0.000, E1   +75.680, E3 +8497.826}
SPL {X  -152.710, Y  +324.020, Z    +0.000, E1   +75.365, E3 +8507.308}
SPL {X  -139.497, Y  +296.529, Z    +0.000, E1   +77.231, E3 +8500.880}
ENDSPLINE

SPLINE
SPL {X  -139.520, Y  +296.568, Z    +0.000, E1   +75.884, E3 +8513.527}
ENDSPLINE

SPLINE
SPL {X  -138.554, Y  +294.984, Z    +0.000, E1   +74.772, E3 +8523.408}
SPL {X  -137.186, Y  +292.805, Z    +0.000, E1   +73.993, E3 +8530.648}
SPL {X  -133.270, Y  +286.961, Z    +0.000, E1   +73.739, E3 +8535.362}
SPL {X  -129.057, Y  +281.230, Z    +0.000, E1   +73.118, E3 +8542.269}
SPL {X  -124.650, Y  +275.749, Z    +0.000, E1   +72.674, E3 +8547.302}
SPL {X  -121.687, Y  +272.322, Z    +0.000, E1   +72.100, E3 +8551.611}
SPL {X  -113.980, Y  +264.229, Z    +0.000, E1   +74.120, E3 +8547.750}
SPL {X   -56.216, Y  +227.692, Z    +0.000, E1   +56.267, E3 +8724.474}
ENDSPLINE

SPLINE
SPL {X  -126.995, Y  +278.604, Z    +0.000, E1   +59.937, E3 +8896.714}
SPL {X  -150.196, Y  +317.640, Z    +0.000, E1   +49.956, E3 +8905.169}
SPL {X  -157.261, Y  +338.316, Z    +0.000, E1   +40.017, E3 +8906.864}
SPL {X  -160.924, Y  +355.726, Z    +0.000, E1   +27.715, E3 +8907.305}
SPL {X  -162.423, Y  +369.141, Z    +0.000, E1   +15.207, E3 +8907.740}
SPL {X  -162.811, Y  +378.755, Z    +0.000, E1    +4.616, E3 +8907.655}
SPL {X  -162.820, Y  +382.684, Z    +0.000, E1    -0.227, E3 +8907.209}
SPL {X  -162.820, Y  +387.227, Z    +0.000, E1   -12.320, E3 +8906.964}
SPL {X  -162.820, Y  +392.558, Z    +0.000, E1   -27.778, E3 +8907.000}
SPL {X  -162.820, Y  +400.474, Z    +0.000, E1   -46.251, E3 +8906.864}
SPL {X  -162.820, Y  +414.510, Z    +0.000, E1   -65.115, E3 +8906.307}
SPL {X  -162.820, Y  +465.064, Z    +0.000, E1   -76.269, E3 +8916.155}
SPL {X  -157.184, Y  +715.968, Z    +0.000, E1   -76.600, E3 +9012.112}
SPL {X  -156.461, Y  +718.560, Z    +0.000, E1   -75.553, E3 +9025.532}
SPL {X  -151.911, Y  +732.096, Z    +0.000, E1   -75.235, E3 +9036.086}
SPL {X  -146.569, Y  +744.407, Z    +0.000, E1   -74.677, E3 +9047.891}
SPL {X  -142.375, Y  +752.491, Z    +0.000, E1   -74.335, E3 +9054.918}
SPL {X  -139.539, Y  +757.399, Z    +0.000, E1   -73.892, E3 +9061.116}
SPL {X  -136.017, Y  +762.997, Z    +0.000, E1   -73.579, E3 +9066.298}
SPL {X  -133.089, Y  +767.296, Z    +0.000, E1   -73.251, E3 +9070.756}
SPL {X  -129.985, Y  +771.553, Z    +0.000, E1   -72.801, E3 +9075.750}
SPL {X  -126.581, Y  +775.909, Z    +0.000, E1   -72.426, E3 +9080.061}
SPL {X  -123.329, Y  +779.803, Z    +0.000, E1   -71.936, E3 +9084.443}
SPL {X  -119.291, Y  +784.315, Z    +0.000, E1   -72.148, E3 +9085.855}
SPL {X   -57.587, Y  +825.796, Z    +0.000, E1   -56.753, E3 +9239.617}
ENDSPLINE

SPLINE
SPL {X  -124.075, Y  +778.932, Z    +0.000, E1   -61.393, E3 +9433.246}
SPL {X  -147.028, Y  +743.450, Z    +0.000, E1   -53.078, E3 +9439.983}
SPL {X  -152.552, Y  +730.406, Z    +0.000, E1   -48.136, E3 +9441.401}
SPL {X  -159.377, Y  +706.804, Z    +0.000, E1   -34.828, E3 +9442.569}
SPL {X  -162.134, Y  +688.425, Z    +0.000, E1   -19.100, E3 +9442.506}
SPL {X  -162.803, Y  +675.871, Z    +0.000, E1    -5.469, E3 +9442.690}
SPL {X  -162.820, Y  +671.500, Z    +0.000, E1    +0.000, E3 +9442.258}
SPL {X  -162.820, Y  +669.743, Z    +0.000, E1    +4.352, E3 +9442.053}
SPL {X  -162.820, Y  +665.917, Z    +0.000, E1   +15.272, E3 +9442.048}
SPL {X  -162.820, Y  +661.245, Z    +0.000, E1   +28.879, E3 +9441.889}
SPL {X  -162.820, Y  +654.015, Z    +0.000, E1   +45.814, E3 +9442.036}
SPL {X  -162.820, Y  +641.345, Z    +0.000, E1   +63.138, E3 +9442.083}
SPL {X  -162.820, Y  +620.039, Z    +0.000, E1   +75.979, E3 +9440.693}
SPL {X  -162.820, Y  +571.094, Z    +0.000, E1   +77.089, E3 +9455.872}
SPL {X  -157.487, Y  +339.169, Z    +0.000, E1   +76.425, E3 +9548.975}
SPL {X  -156.386, Y  +335.181, Z    +0.000, E1   +75.555, E3 +9561.036}
SPL {X  -152.710, Y  +324.020, Z    +0.000, E1   +75.365, E3 +9568.847}
SPL {X  -139.497, Y  +296.529, Z    +0.000, E1   +77.231, E3 +9562.418}
ENDSPLINE

SPLINE
SPL {X  -139.792, Y  +297.022, Z    +0.000, E1   +76.273, E3 +9571.113}
ENDSPLINE

SPLINE
SPL {X  -138.933, Y  +295.600, Z    +0.000, E1   +75.173, E3 +9581.596}
SPL {X  -137.186, Y  +292.805, Z    +0.000, E1   +73.993, E3 +9592.187}
SPL {X  -133.270, Y  +286.961, Z    +0.000, E1   +73.739, E3 +9596.900}
SPL {X  -130.283, Y  +282.844, Z    +0.000, E1   +73.297, E3 +9601.792}
SPL {X  -126.880, Y  +278.461, Z    +0.000, E1   +72.855, E3 +9606.542}
SPL {X  -123.363, Y  +274.237, Z    +0.000, E1   +72.376, E3 +9611.024}
SPL {X  -121.018, Y  +271.573, Z    +0.000, E1   +72.049, E3 +9613.710}
SPL {X  -113.980, Y  +264.229, Z    +0.000, E1   +74.120, E3 +9609.288}
SPL {X   -56.216, Y  +227.692, Z    +0.000, E1   +56.267, E3 +9786.012}
ENDSPLINE

SPLINE
SPL {X  -126.995, Y  +278.604, Z    +0.000, E1   +59.937, E3 +9958.252}
SPL {X  -150.196, Y  +317.640, Z    +0.000, E1   +49.956, E3 +9966.707}
SPL {X  -157.261, Y  +338.316, Z    +0.000, E1   +40.017, E3 +9968.402}
SPL {X  -160.924, Y  +355.726, Z    +0.000, E1   +27.715, E3 +9968.843}
SPL {X  -162.423, Y  +369.141, Z    +0.000, E1   +15.207, E3 +9969.279}
SPL {X  -162.811, Y  +378.755, Z    +0.000, E1    +4.616, E3 +9969.193}
SPL {X  -162.820, Y  +382.684, Z    +0.000, E1    -0.227, E3 +9968.748}
SPL {X  -162.820, Y  +387.227, Z    +0.000, E1   -12.320, E3 +9968.502}
SPL {X  -162.820, Y  +392.558, Z    +0.000, E1   -27.778, E3 +9968.539}
SPL {X  -162.820, Y  +398.468, Z    +0.000, E1   -42.446, E3 +9968.389}
SPL {X  -162.820, Y  +404.415, Z    +0.000, E1   -53.236, E3 +9968.428}
SPL {X  -162.820, Y  +414.510, Z    +0.000, E1   -65.115, E3 +9967.845}
SPL {X  -162.820, Y  +465.064, Z    +0.000, E1   -76.269, E3 +9977.693}
SPL {X  -157.184, Y  +715.968, Z    +0.000, E1   -76.600, E3 +10073.651}
SPL {X  -156.461, Y  +718.560, Z    +0.000, E1   -75.553, E3 +10087.071}
SPL {X  -151.911, Y  +732.096, Z    +0.000, E1   -75.235, E3 +10097.625}
SPL {X  -146.569, Y  +744.407, Z    +0.000, E1   -74.677, E3 +10109.429}
SPL {X  -142.375, Y  +752.491, Z    +0.000, E1   -74.335, E3 +10116.456}
SPL {X  -139.539, Y  +757.399, Z    +0.000, E1   -73.892, E3 +10122.654}
SPL {X  -136.017, Y  +762.997, Z    +0.000, E1   -73.579, E3 +10127.836}
SPL {X  -133.089, Y  +767.296, Z    +0.000, E1   -73.251, E3 +10132.294}
SPL {X  -129.985, Y  +771.553, Z    +0.000, E1   -72.801, E3 +10137.288}
SPL {X  -126.581, Y  +775.909, Z    +0.000, E1   -72.426, E3 +10141.599}
SPL {X  -123.329, Y  +779.803, Z    +0.000, E1   -71.936, E3 +10145.981}
SPL {X  -119.291, Y  +784.315, Z    +0.000, E1   -72.148, E3 +10147.393}
SPL {X   -57.587, Y  +825.796, Z    +0.000, E1   -56.753, E3 +10301.156}
ENDSPLINE

SPLINE
SPL {X  -124.075, Y  +778.932, Z    +0.000, E1   -61.393, E3 +10494.785}
SPL {X  -147.028, Y  +743.450, Z    +0.000, E1   -53.078, E3 +10501.522}
SPL {X  -152.552, Y  +730.406, Z    +0.000, E1   -48.136, E3 +10502.939}
SPL {X  -159.377, Y  +706.804, Z    +0.000, E1   -34.828, E3 +10504.107}
SPL {X  -162.134, Y  +688.425, Z    +0.000, E1   -19.100, E3 +10504.044}
SPL {X  -162.803, Y  +675.871, Z    +0.000, E1    -5.469, E3 +10504.228}
SPL {X  -162.820, Y  +671.500, Z    +0.000, E1    +0.000, E3 +10503.796}
SPL {X  -162.820, Y  +669.743, Z    +0.000, E1    +4.352, E3 +10503.592}
SPL {X  -162.820, Y  +665.917, Z    +0.000, E1   +15.272, E3 +10503.586}
SPL {X  -162.820, Y  +661.245, Z    +0.000, E1   +28.879, E3 +10503.427}
SPL {X  -162.820, Y  +654.015, Z    +0.000, E1   +45.814, E3 +10503.574}
SPL {X  -162.820, Y  +641.345, Z    +0.000, E1   +63.138, E3 +10503.622}
SPL {X  -162.820, Y  +620.039, Z    +0.000, E1   +75.979, E3 +10502.231}
SPL {X  -162.820, Y  +571.094, Z    +0.000, E1   +77.089, E3 +10517.410}
SPL {X  -158.110, Y  +341.619, Z    +0.000, E1   +77.339, E3 +10599.060}
SPL {X  -156.597, Y  +335.917, Z    +0.000, E1   +75.680, E3 +10620.903}
SPL {X  -152.710, Y  +324.020, Z    +0.000, E1   +75.365, E3 +10630.385}
SPL {X  -139.497, Y  +296.529, Z    +0.000, E1   +77.231, E3 +10623.957}
ENDSPLINE

SPLINE
SPL {X  -139.792, Y  +297.022, Z    +0.000, E1   +76.273, E3 +10632.652}
ENDSPLINE

SPLINE
SPL {X  -138.933, Y  +295.600, Z    +0.000, E1   +75.173, E3 +10643.135}
SPL {X  -137.186, Y  +292.805, Z    +0.000, E1   +73.993, E3 +10653.725}
SPL {X  -133.270, Y  +286.961, Z    +0.000, E1   +73.739, E3 +10658.438}
SPL {X  -130.283, Y  +282.844, Z    +0.000, E1   +73.297, E3 +10663.330}
SPL {X  -127.795, Y  +279.610, Z    +0.000, E1   +72.860, E3 +10667.461}
SPL {X  -124.650, Y  +275.749, Z    +0.000, E1   +72.674, E3 +10670.379}
SPL {X  -121.687, Y  +272.322, Z    +0.000, E1   +72.100, E3 +10674.688}
SPL {X  -113.980, Y  +264.229, Z    +0.000, E1   +74.120, E3 +10670.826}
SPL {X   -56.216, Y  +227.692, Z    +0.000, E1   +56.267, E3 +10847.550}
ENDSPLINE

SPLINE
SPL {X  -126.995, Y  +278.604, Z    +0.000, E1   +59.937, E3 +11019.791}
SPL {X  -150.196, Y  +317.640, Z    +0.000, E1   +49.956, E3 +11028.246}
SPL {X  -157.261, Y  +338.316, Z    +0.000, E1   +40.017, E3 +11029.941}
SPL {X  -160.924, Y  +355.726, Z    +0.000, E1   +27.715, E3 +11030.382}
SPL {X  -162.423, Y  +369.141, Z    +0.000, E1   +15.207, E3 +11030.817}
SPL {X  -162.811, Y  +378.755, Z    +0.000, E1    +4.616, E3 +11030.732}
SPL {X  -162.820, Y  +382.684, Z    +0.000, E1    -0.227, E3 +11030.286}
SPL {X  -162.820, Y  +387.227, Z    +0.000, E1   -12.320, E3 +11030.041}
SPL {X  -162.820, Y  +392.558, Z    +0.000, E1   -27.778, E3 +11030.077}
SPL {X  -162.820, Y  +400.474, Z    +0.000, E1   -46.251, E3 +11029.941}
SPL {X  -162.820, Y  +414.510, Z    +0.000, E1   -65.115, E3 +11029.384}
SPL {X  -162.820, Y  +465.064, Z    +0.000, E1   -76.269, E3 +11039.232}
SPL {X  -157.184, Y  +715.968, Z    +0.000, E1   -76.600, E3 +11135.189}
SPL {X  -156.461, Y  +718.560, Z    +0.000, E1   -75.553, E3 +11148.609}
SPL {X  -151.911, Y  +732.096, Z    +0.000, E1   -75.235, E3 +11159.163}
SPL {X  -146.569, Y  +744.407, Z    +0.000, E1   -74.677, E3 +11170.967}
SPL {X  -142.375, Y  +752.491, Z    +0.000, E1   -74.335, E3 +11177.995}
SPL {X  -139.539, Y  +757.399, Z    +0.000, E1   -73.892, E3 +11184.192}
SPL {X  -136.017, Y  +762.997, Z    +0.000, E1   -73.579, E3 +11189.375}
SPL {X  -133.089, Y  +767.296, Z    +0.000, E1   -73.251, E3 +11193.833}
SPL {X  -129.985, Y  +771.553, Z    +0.000, E1   -72.801, E3 +11198.827}
SPL {X  -126.581, Y  +775.909, Z    +0.000, E1   -72.426, E3 +11203.138}
SPL {X  -123.329, Y  +779.803, Z    +0.000, E1   -71.936, E3 +11207.520}
SPL {X  -119.291, Y  +784.315, Z    +0.000, E1   -72.148, E3 +11208.932}
SPL {X   -57.587, Y  +825.796, Z    +0.000, E1   -56.753, E3 +11362.694}
ENDSPLINE

SPLINE
SPL {X  -124.075, Y  +778.932, Z    +0.000, E1   -61.393, E3 +11556.323}
SPL {X  -147.028, Y  +743.450, Z    +0.000, E1   -53.078, E3 +11563.060}
SPL {X  -152.552, Y  +730.406, Z    +0.000, E1   -48.136, E3 +11564.478}
SPL {X  -159.377, Y  +706.804, Z    +0.000, E1   -34.828, E3 +11565.646}
SPL {X  -162.134, Y  +688.425, Z    +0.000, E1   -19.100, E3 +11565.583}
SPL {X  -162.803, Y  +675.871, Z    +0.000, E1    -5.469, E3 +11565.766}
SPL {X  -162.820, Y  +671.500, Z    +0.000, E1    +0.000, E3 +11565.335}
SPL {X  -162.820, Y  +669.743, Z    +0.000, E1    +4.352, E3 +11565.130}
SPL {X  -162.820, Y  +665.917, Z    +0.000, E1   +15.272, E3 +11565.125}
SPL {X  -162.820, Y  +661.245, Z    +0.000, E1   +28.879, E3 +11564.966}
SPL {X  -162.820, Y  +654.015, Z    +0.000, E1   +45.814, E3 +11565.113}
SPL {X  -162.820, Y  +641.345, Z    +0.000, E1   +63.138, E3 +11565.160}
SPL {X  -162.820, Y  +620.039, Z    +0.000, E1   +75.979, E3 +11563.770}
SPL {X  -162.820, Y  +571.094, Z    +0.000, E1   +77.089, E3 +11578.948}
SPL {X  -157.487, Y  +339.169, Z    +0.000, E1   +76.425, E3 +11672.052}
SPL {X  -156.386, Y  +335.181, Z    +0.000, E1   +75.555, E3 +11684.113}
SPL {X  -152.710, Y  +324.020, Z    +0.000, E1   +75.365, E3 +11691.924}
SPL {X  -139.497, Y  +296.529, Z    +0.000, E1   +77.231, E3 +11685.495}
ENDSPLINE

SPLINE
SPL {X  -139.792, Y  +297.022, Z    +0.000, E1   +76.273, E3 +11694.190}
ENDSPLINE

SPLINE
SPL {X  -138.933, Y  +295.600, Z    +0.000, E1   +75.173, E3 +11704.673}
SPL {X  -137.186, Y  +292.805, Z    +0.000, E1   +73.993, E3 +11715.264}
SPL {X  -133.270, Y  +286.961, Z    +0.000, E1   +73.739, E3 +11719.977}
SPL {X  -130.283, Y  +282.844, Z    +0.000, E1   +73.297, E3 +11724.869}
SPL {X  -126.880, Y  +278.461, Z    +0.000, E1   +72.855, E3 +11729.619}
SPL {X  -123.363, Y  +274.237, Z    +0.000, E1   +72.376, E3 +11734.101}
SPL {X  -121.018, Y  +271.573, Z    +0.000, E1   +72.049, E3 +11736.787}
SPL {X  -113.980, Y  +264.229, Z    +0.000, E1   +74.120, E3 +11732.365}
SPL {X   -56.216, Y  +227.692, Z    +0.000, E1   +56.267, E3 +11909.089}
ENDSPLINE

SPLINE
SPL {X  -126.995, Y  +278.604, Z    +0.000, E1   +59.937, E3 +12081.329}
SPL {X  -150.196, Y  +317.640, Z    +0.000, E1   +49.956, E3 +12089.784}
SPL {X  -157.261, Y  +338.316, Z    +0.000, E1   +40.017, E3 +12091.479}
SPL {X  -160.924, Y  +355.726, Z    +0.000, E1   +27.715, E3 +12091.920}
SPL {X  -162.423, Y  +369.141, Z    +0.000, E1   +15.207, E3 +12092.356}
SPL {X  -162.811, Y  +378.755, Z    +0.000, E1    +4.616, E3 +12092.270}
SPL {X  -162.820, Y  +382.684, Z    +0.000, E1    -0.227, E3 +12091.825}
SPL {X  -162.820, Y  +385.721, Z    +0.000, E1    -8.371, E3 +12091.640}
SPL {X  -162.820, Y  +388.532, Z    +0.000, E1   -16.412, E3 +12091.527}
SPL {X  -162.820, Y  +392.558, Z    +0.000, E1   -27.778, E3 +12091.616}
SPL {X  -162.820, Y  +400.474, Z    +0.000, E1   -46.251, E3 +12091.479}
SPL {X  -162.820, Y  +414.510, Z    +0.000, E1   -65.115, E3 +12090.922}
SPL {X  -162.820, Y  +465.064, Z    +0.000, E1   -76.269, E3 +12100.770}
SPL {X  -157.184, Y  +715.968, Z    +0.000, E1   -76.600, E3 +12196.728}
SPL {X  -156.461, Y  +718.560, Z    +0.000, E1   -75.553, E3 +12210.148}
SPL {X  -151.911, Y  +732.096, Z    +0.000, E1   -75.235, E3 +12220.702}
SPL {X  -146.569, Y  +744.407, Z    +0.000, E1   -74.677, E3 +12232.506}
SPL {X  -142.375, Y  +752.491, Z    +0.000, E1   -74.335, E3 +12239.533}
SPL {X  -139.539, Y  +757.399, Z    +0.000, E1   -73.892, E3 +12245.731}
SPL {X  -136.017, Y  +762.997, Z    +0.000, E1   -73.579, E3 +12250.913}
SPL {X  -133.089, Y  +767.296, Z    +0.000, E1   -73.251, E3 +12255.371}
SPL {X  -129.985, Y  +771.553, Z    +0.000, E1   -72.801, E3 +12260.365}
SPL {X  -126.581, Y  +775.909, Z    +0.000, E1   -72.426, E3 +12264.676}
SPL {X  -123.329, Y  +779.803, Z    +0.000, E1   -71.936, E3 +12269.058}
SPL {X  -119.291, Y  +784.315, Z    +0.000, E1   -72.148, E3 +12270.470}
SPL {X   -57.587, Y  +825.796, Z    +0.000, E1   -56.753, E3 +12424.233}
ENDSPLINE

SPLINE
SPL {X  -124.075, Y  +778.932, Z    +0.000, E1   -61.393, E3 +12617.862}
SPL {X  -147.028, Y  +743.450, Z    +0.000, E1   -53.078, E3 +12624.599}
SPL {X  -152.552, Y  +730.406, Z    +0.000, E1   -48.136, E3 +12626.016}
SPL {X  -159.377, Y  +706.804, Z    +0.000, E1   -34.828, E3 +12627.184}
SPL {X  -162.134, Y  +688.425, Z    +0.000, E1   -19.100, E3 +12627.121}
SPL {X  -162.803, Y  +675.871, Z    +0.000, E1    -5.469, E3 +12627.305}
SPL {X  -162.820, Y  +671.500, Z    +0.000, E1    +0.000, E3 +12626.873}
SPL {X  -162.820, Y  +669.743, Z    +0.000, E1    +4.352, E3 +12626.669}
SPL {X  -162.820, Y  +665.917, Z    +0.000, E1   +15.272, E3 +12626.663}
SPL {X  -162.820, Y  +661.245, Z    +0.000, E1   +28.879, E3 +12626.504}
SPL {X  -162.820, Y  +654.015, Z    +0.000, E1   +45.814, E3 +12626.651}
SPL {X  -162.820, Y  +641.345, Z    +0.000, E1   +63.138, E3 +12626.698}
SPL {X  -162.820, Y  +620.039, Z    +0.000, E1   +75.979, E3 +12625.308}
SPL {X  -162.820, Y  +571.094, Z    +0.000, E1   +77.089, E3 +12640.487}
SPL {X  -157.487, Y  +339.169, Z    +0.000, E1   +76.425, E3 +12733.591}
SPL {X  -156.386, Y  +335.181, Z    +0.000, E1   +75.555, E3 +12745.652}
SPL {X  -152.710, Y  +324.020, Z    +0.000, E1   +75.365, E3 +12753.462}
SPL {X  -139.497, Y  +296.529, Z    +0.000, E1   +77.231, E3 +12747.034}
ENDSPLINE

SPLINE
SPL {X  -139.792, Y  +297.022, Z    +0.000, E1   +76.273, E3 +12755.729}
ENDSPLINE

SPLINE
SPL {X  -138.933, Y  +295.600, Z    +0.000, E1   +75.173, E3 +12766.212}
SPL {X  -137.186, Y  +292.805, Z    +0.000, E1   +73.993, E3 +12776.802}
SPL {X  -133.270, Y  +286.961, Z    +0.000, E1   +73.739, E3 +12781.515}
SPL {X  -130.283, Y  +282.844, Z    +0.000, E1   +73.297, E3 +12786.407}
SPL {X  -127.795, Y  +279.610, Z    +0.000, E1   +72.860, E3 +12790.537}
SPL {X  -124.650, Y  +275.749, Z    +0.000, E1   +72.674, E3 +12793.456}
SPL {X  -121.687, Y  +272.322, Z    +0.000, E1   +72.100, E3 +12797.765}
SPL {X  -113.980, Y  +264.229, Z    +0.000, E1   +74.120, E3 +12793.903}
SPL {X   -56.216, Y  +227.692, Z    +0.000, E1   +56.267, E3 +12970.627}
ENDSPLINE

SPLINE
SPL {X  -126.995, Y  +278.604, Z    +0.000, E1   +59.937, E3 +13142.868}
SPL {X  -150.196, Y  +317.640, Z    +0.000, E1   +49.956, E3 +13151.323}
SPL {X  -157.261, Y  +338.316, Z    +0.000, E1   +40.017, E3 +13153.018}
SPL {X  -160.924, Y  +355.726, Z    +0.000, E1   +27.715, E3 +13153.459}
SPL {X  -162.423, Y  +369.141, Z    +0.000, E1   +15.207, E3 +13153.894}
SPL {X  -162.811, Y  +378.755, Z    +0.000, E1    +4.616, E3 +13153.808}
SPL {X  -162.820, Y  +382.684, Z    +0.000, E1    -0.227, E3 +13153.363}
SPL {X  -162.820, Y  +387.227, Z    +0.000, E1   -12.320, E3 +13153.118}
SPL {X  -162.820, Y  +392.558, Z    +0.000, E1   -27.778, E3 +13153.154}
SPL {X  -162.820, Y  +400.474, Z    +0.000, E1   -46.251, E3 +13153.018}
SPL {X  -162.820, Y  +414.510, Z    +0.000, E1   -65.115, E3 +13152.461}
SPL {X  -162.820, Y  +465.064, Z    +0.000, E1   -76.269, E3 +13162.309}
SPL {X  -157.184, Y  +715.968, Z    +0.000, E1   -76.600, E3 +13258.266}
SPL {X  -156.461, Y  +718.560, Z    +0.000, E1   -75.553, E3 +13271.686}
SPL {X  -153.015, Y  +729.150, Z    +0.000, E1   -75.312, E3 +13279.775}
SPL {X  -149.053, Y  +739.025, Z    +0.000, E1   -74.952, E3 +13288.571}
SPL {X  -145.525, Y  +746.527, Z    +0.000, E1   -74.526, E3 +13296.364}
SPL {X  -142.375, Y  +752.491, Z    +0.000, E1   -74.335, E3 +13301.072}
SPL {X  -139.539, Y  +757.399, Z    +0.000, E1   -73.892, E3 +13307.269}
SPL {X  -136.017, Y  +762.997, Z    +0.000, E1   -73.579, E3 +13312.452}
SPL {X  -133.089, Y  +767.296, Z    +0.000, E1   -73.251, E3 +13316.910}
SPL {X  -129.985, Y  +771.553, Z    +0.000, E1   -72.801, E3 +13321.904}
SPL {X  -126.581, Y  +775.909, Z    +0.000, E1   -72.426, E3 +13326.215}
SPL {X  -123.329, Y  +779.803, Z    +0.000, E1   -71.936, E3 +13330.597}
SPL {X  -119.291, Y  +784.315, Z    +0.000, E1   -72.148, E3 +13332.009}
SPL {X   -57.587, Y  +825.796, Z    +0.000, E1   -56.753, E3 +13485.771}
ENDSPLINE

SPLINE
SPL {X  -124.075, Y  +778.932, Z    +0.000, E1   -61.393, E3 +13679.400}
SPL {X  -150.653, Y  +735.257, Z    +0.000, E1   -50.160, E3 +13687.079}
SPL {X  -159.377, Y  +706.804, Z    +0.000, E1   -34.828, E3 +13688.723}
SPL {X  -162.134, Y  +688.425, Z    +0.000, E1   -19.100, E3 +13688.659}
SPL {X  -162.803, Y  +675.871, Z    +0.000, E1    -5.469, E3 +13688.843}
SPL {X  -162.820, Y  +671.500, Z    +0.000, E1    +0.000, E3 +13688.411}
SPL {X  -162.820, Y  +669.743, Z    +0.000, E1    +4.352, E3 +13688.207}
SPL {X  -162.820, Y  +665.917, Z    +0.000, E1   +15.272, E3 +13688.202}
SPL {X  -162.820, Y  +661.245, Z    +0.000, E1   +28.879, E3 +13688.043}
SPL {X  -162.820, Y  +654.015, Z    +0.000, E1   +45.814, E3 +13688.190}
SPL {X  -162.820, Y  +641.345, Z    +0.000, E1   +63.138, E3 +13688.237}
SPL {X  -162.820, Y  +620.039, Z    +0.000, E1   +75.979, E3 +13686.847}
SPL {X  -162.820, Y  +578.479, Z    +0.000, E1   +77.260, E3 +13699.117}
SPL {X  -162.820, Y  +557.052, Z    +0.000, E1   +76.772, E3 +13707.599}
SPL {X  -157.487, Y  +339.169, Z    +0.000, E1   +76.425, E3 +13795.129}
SPL {X  -156.386, Y  +335.181, Z    +0.000, E1   +75.555, E3 +13807.190}
SPL {X  -152.710, Y  +324.020, Z    +0.000, E1   +75.365, E3 +13815.000}
SPL {X  -139.497, Y  +296.529, Z    +0.000, E1   +77.231, E3 +13808.572}
ENDSPLINE

SPLINE
SPL {X  -139.792, Y  +297.022, Z    +0.000, E1   +76.273, E3 +13817.267}
ENDSPLINE

SPLINE
SPL {X  -138.933, Y  +295.600, Z    +0.000, E1   +75.173, E3 +13827.750}
SPL {X  -137.186, Y  +292.805, Z    +0.000, E1   +73.993, E3 +13838.340}
SPL {X  -133.270, Y  +286.961, Z    +0.000, E1   +73.739, E3 +13843.054}
SPL {X  -130.283, Y  +282.844, Z    +0.000, E1   +73.297, E3 +13847.946}
SPL {X  -126.880, Y  +278.461, Z    +0.000, E1   +72.855, E3 +13852.696}
SPL {X  -124.135, Y  +275.140, Z    +0.000, E1   +72.554, E3 +13855.825}
SPL {X  -121.687, Y  +272.322, Z    +0.000, E1   +72.100, E3 +13859.304}
SPL {X  -113.980, Y  +264.229, Z    +0.000, E1   +74.120, E3 +13855.442}
SPL {X   -56.216, Y  +227.692, Z    +0.000, E1   +56.267, E3 +14032.166}
ENDSPLINE

SPLINE
SPL {X  -126.995, Y  +278.604, Z    +0.000, E1   +59.937, E3 +14204.406}
SPL {X  -150.196, Y  +317.640, Z    +0.000, E1   +49.956, E3 +14212.861}
SPL {X  -157.261, Y  +338.316, Z    +0.000, E1   +40.017, E3 +14214.556}
SPL {X  -160.924, Y  +355.726, Z    +0.000, E1   +27.715, E3 +14214.997}
SPL {X  -162.423, Y  +369.141, Z    +0.000, E1   +15.207, E3 +14215.432}
SPL {X  -162.811, Y  +378.755, Z    +0.000, E1    +4.616, E3 +14215.347}
SPL {X  -162.820, Y  +382.684, Z    +0.000, E1    -0.227, E3 +14214.902}
SPL {X  -162.820, Y  +385.721, Z    +0.000, E1    -8.371, E3 +14214.717}
SPL {X  -162.820, Y  +388.532, Z    +0.000, E1   -16.412, E3 +14214.604}
SPL {X  -162.820, Y  +392.558, Z    +0.000, E1   -27.778, E3 +14214.692}
SPL {X  -162.820, Y  +400.474, Z    +0.000, E1   -46.251, E3 +14214.556}
SPL {X  -162.820, Y  +414.510, Z    +0.000, E1   -65.115, E3 +14213.999}
SPL {X  -162.820, Y  +465.064, Z    +0.000, E1   -76.269, E3 +14223.847}
SPL {X  -157.184, Y  +715.968, Z    +0.000, E1   -76.600, E3 +14319.805}
SPL {X  -156.461, Y  +718.560, Z    +0.000, E1   -75.553, E3 +14333.225}
SPL {X  -153.015, Y  +729.150, Z    +0.000, E1   -75.312, E3 +14341.314}
SPL {X  -149.053, Y  +739.025, Z    +0.000, E1   -74.952, E3 +14350.109}
SPL {X  -144.053, Y  +749.389, Z    +0.000, E1   -74.457, E3 +14360.101}
SPL {X  -139.539, Y  +757.399, Z    +0.000, E1   -73.892, E3 +14368.808}
SPL {X  -136.017, Y  +762.997, Z    +0.000, E1   -73.579, E3 +14373.990}
SPL {X  -133.089, Y  +767.296, Z    +0.000, E1   -73.251, E3 +14378.448}
SPL {X  -129.985, Y  +771.553, Z    +0.000, E1   -72.801, E3 +14383.442}
SPL {X  -126.581, Y  +775.909, Z    +0.000, E1   -72.426, E3 +14387.753}
SPL {X  -123.329, Y  +779.803, Z    +0.000, E1   -71.936, E3 +14392.135}
SPL {X  -119.291, Y  +784.315, Z    +0.000, E1   -72.148, E3 +14393.547}
SPL {X   -57.587, Y  +825.796, Z    +0.000, E1   -56.753, E3 +14547.309}
ENDSPLINE

SPLINE
SPL {X  -124.075, Y  +778.932, Z    +0.000, E1   -61.393, E3 +14740.938}
SPL {X  -150.653, Y  +735.257, Z    +0.000, E1   -50.160, E3 +14748.618}
SPL {X  -159.377, Y  +706.804, Z    +0.000, E1   -34.828, E3 +14750.261}
SPL {X  -162.134, Y  +688.425, Z    +0.000, E1   -19.100, E3 +14750.198}
SPL {X  -162.734, Y  +678.779, Z    +0.000, E1    -8.745, E3 +14750.337}
SPL {X  -162.820, Y  +671.589, Z    +0.000, E1    -0.221, E3 +14749.971}
SPL {X  -162.820, Y  +669.743, Z    +0.000, E1    +4.352, E3 +14749.746}
SPL {X  -162.820, Y  +665.917, Z    +0.000, E1   +15.272, E3 +14749.740}
SPL {X  -162.820, Y  +661.245, Z    +0.000, E1   +28.879, E3 +14749.581}
SPL {X  -162.820, Y  +654.015, Z    +0.000, E1   +45.814, E3 +14749.728}
SPL {X  -162.820, Y  +641.345, Z    +0.000, E1   +63.138, E3 +14749.775}
SPL {X  -162.820, Y  +620.039, Z    +0.000, E1   +75.979, E3 +14748.385}
SPL {X  -162.820, Y  +571.094, Z    +0.000, E1   +77.089, E3 +14763.564}
SPL {X  -158.110, Y  +341.619, Z    +0.000, E1   +77.339, E3 +14845.214}
SPL {X  -156.597, Y  +335.917, Z    +0.000, E1   +75.680, E3 +14867.057}
SPL {X  -152.710, Y  +324.020, Z    +0.000, E1   +75.365, E3 +14876.539}
SPL {X  -139.497, Y  +296.529, Z    +0.000, E1   +77.231, E3 +14870.111}
ENDSPLINE

SPLINE
SPL {X  -139.520, Y  +296.568, Z    +0.000, E1   +75.884, E3 +14882.758}
ENDSPLINE

SPLINE
SPL {X  -138.554, Y  +294.984, Z    +0.000, E1   +74.772, E3 +14892.639}
SPL {X  -137.186, Y  +292.805, Z    +0.000, E1   +73.993, E3 +14899.879}
SPL {X  -133.270, Y  +286.961, Z    +0.000, E1   +73.739, E3 +14904.592}
SPL {X  -129.057, Y  +281.230, Z    +0.000, E1   +73.118, E3 +14911.500}
SPL {X  -124.650, Y  +275.749, Z    +0.000, E1   +72.674, E3 +14916.533}
SPL {X  -121.687, Y  +272.322, Z    +0.000, E1   +72.100, E3 +14920.842}
SPL {X  -113.980, Y  +264.229, Z    +0.000, E1   +74.120, E3 +14916.980}
SPL {X   -56.216, Y  +227.692, Z    +0.000, E1   +56.267, E3 +15093.704}
ENDSPLINE

SPLINE
SPL {X  -126.995, Y  +278.604, Z    +0.000, E1   +59.937, E3 +15265.945}
SPL {X  -150.196, Y  +317.640, Z    +0.000, E1   +49.956, E3 +15274.400}
SPL {X  -157.261, Y  +338.316, Z    +0.000, E1   +40.017, E3 +15276.095}
SPL {X  -160.924, Y  +355.726, Z    +0.000, E1   +27.715, E3 +15276.535}
SPL {X  -162.423, Y  +369.141, Z    +0.000, E1   +15.207, E3 +15276.971}
SPL {X  -162.811, Y  +378.755, Z    +0.000, E1    +4.616, E3 +15276.885}
SPL {X  -162.820, Y  +382.684, Z    +0.000, E1    -0.227, E3 +15276.440}
SPL {X  -162.820, Y  +385.721, Z    +0.000, E1    -8.371, E3 +15276.256}
SPL {X  -162.820, Y  +388.532, Z    +0.000, E1   -16.412, E3 +15276.142}
SPL {X  -162.820, Y  +392.558, Z    +0.000, E1   -27.778, E3 +15276.231}
SPL {X  -162.820, Y  +400.474, Z    +0.000, E1   -46.251, E3 +15276.095}
SPL {X  -162.820, Y  +414.510, Z    +0.000, E1   -65.115, E3 +15275.538}
SPL {X  -162.820, Y  +465.064, Z    +0.000, E1   -76.269, E3 +15285.386}
SPL {X  -157.184, Y  +715.968, Z    +0.000, E1   -76.600, E3 +15381.343}
SPL {X  -156.461, Y  +718.560, Z    +0.000, E1   -75.553, E3 +15394.763}
SPL {X  -153.015, Y  +729.150, Z    +0.000, E1   -75.312, E3 +15402.852}
SPL {X  -149.053, Y  +739.025, Z    +0.000, E1   -74.952, E3 +15411.648}
SPL {X  -145.525, Y  +746.527, Z    +0.000, E1   -74.526, E3 +15419.441}
SPL {X  -142.375, Y  +752.491, Z    +0.000, E1   -74.335, E3 +15424.149}
SPL {X  -139.539, Y  +757.399, Z    +0.000, E1   -73.892, E3 +15430.346}
SPL {X  -136.017, Y  +762.997, Z    +0.000, E1   -73.579, E3 +15435.529}
SPL {X  -133.089, Y  +767.296, Z    +0.000, E1   -73.251, E3 +15439.987}
SPL {X  -129.985, Y  +771.553, Z    +0.000, E1   -72.801, E3 +15444.981}
SPL {X  -126.581, Y  +775.909, Z    +0.000, E1   -72.426, E3 +15449.292}
SPL {X  -122.528, Y  +780.725, Z    +0.000, E1   -71.905, E3 +15454.312}
SPL {X  -116.189, Y  +787.563, Z    +0.000, E1   -72.978, E3 +15453.596}
SPL {X   -57.587, Y  +825.796, Z    +0.000, E1   -56.753, E3 +15608.848}
ENDSPLINE

SPLINE
SPL {X  -124.075, Y  +778.932, Z    +0.000, E1   -61.393, E3 +15802.477}
SPL {X  -147.028, Y  +743.450, Z    +0.000, E1   -53.078, E3 +15809.214}
SPL {X  -152.552, Y  +730.406, Z    +0.000, E1   -48.136, E3 +15810.632}
SPL {X  -159.377, Y  +706.804, Z    +0.000, E1   -34.828, E3 +15811.800}
SPL {X  -162.134, Y  +688.425, Z    +0.000, E1   -19.100, E3 +15811.736}
SPL {X  -162.803, Y  +675.871, Z    +0.000, E1    -5.469, E3 +15811.920}
SPL {X  -162.820, Y  +671.500, Z    +0.000, E1    +0.000, E3 +15811.488}
SPL {X  -162.820, Y  +669.743, Z    +0.000, E1    +4.352, E3 +15811.284}
SPL {X  -162.820, Y  +665.917, Z    +0.000, E1   +15.272, E3 +15811.279}
SPL {X  -162.820, Y  +661.245, Z    +0.000, E1   +28.879, E3 +15811.120}
SPL {X  -162.820, Y  +654.015, Z    +0.000, E1   +45.814, E3 +15811.267}
SPL {X  -162.820, Y  +641.345, Z    +0.000, E1   +63.138, E3 +15811.314}
SPL {X  -162.820, Y  +620.039, Z    +0.000, E1   +75.979, E3 +15809.924}
SPL {X  -162.820, Y  +571.094, Z    +0.000, E1   +77.089, E3 +15825.102}
SPL {X  -157.487, Y  +339.169, Z    +0.000, E1   +76.425, E3 +15918.206}
SPL {X  -156.386, Y  +335.181, Z    +0.000, E1   +75.555, E3 +15930.267}
SPL {X  -152.710, Y  +324.020, Z    +0.000, E1   +75.365, E3 +15938.077}
SPL {X  -139.497, Y  +296.529, Z    +0.000, E1   +77.231, E3 +15931.649}
ENDSPLINE

SPLINE
SPL {X  -139.520, Y  +296.568, Z    +0.000, E1   +75.884, E3 +15944.296}
ENDSPLINE

SPLINE
SPL {X  -138.554, Y  +294.984, Z    +0.000, E1   +74.772, E3 +15954.177}
SPL {X  -137.186, Y  +292.805, Z    +0.000, E1   +73.993, E3 +15961.417}
SPL {X  -133.270, Y  +286.961, Z    +0.000, E1   +73.739, E3 +15966.131}
SPL {X  -130.283, Y  +282.844, Z    +0.000, E1   +73.297, E3 +15971.023}
SPL {X  -127.795, Y  +279.610, Z    +0.000, E1   +72.860, E3 +15975.153}
SPL {X  -124.650, Y  +275.749, Z    +0.000, E1   +72.674, E3 +15978.071}
SPL {X  -121.687, Y  +272.322, Z    +0.000, E1   +72.100, E3 +15982.381}
SPL {X  -113.980, Y  +264.229, Z    +0.000, E1   +74.120, E3 +15978.519}
SPL {X   -56.216, Y  +227.692, Z    +0.000, E1   +56.267, E3 +16155.243}
ENDSPLINE

SPLINE
SPL {X  -126.995, Y  +278.604, Z    +0.000, E1   +59.937, E3 +16327.483}
SPL {X  -150.196, Y  +317.640, Z    +0.000, E1   +49.956, E3 +16335.938}
SPL {X  -157.261, Y  +338.316, Z    +0.000, E1   +40.017, E3 +16337.633}
SPL {X  -160.924, Y  +355.726, Z    +0.000, E1   +27.715, E3 +16338.074}
SPL {X  -162.423, Y  +369.141, Z    +0.000, E1   +15.207, E3 +16338.509}
SPL {X  -162.811, Y  +378.755, Z    +0.000, E1    +4.616, E3 +16338.424}
SPL {X  -162.820, Y  +382.684, Z    +0.000, E1    -0.227, E3 +16337.978}
SPL {X  -162.820, Y  +387.227, Z    +0.000, E1   -12.320, E3 +16337.733}
SPL {X  -162.820, Y  +392.558, Z    +0.000, E1   -27.778, E3 +16337.769}
SPL {X  -162.820, Y  +400.474, Z    +0.000, E1   -46.251, E3 +16337.633}
SPL {X  -162.820, Y  +414.510, Z    +0.000, E1   -65.115, E3 +16337.076}
SPL {X  -162.820, Y  +465.064, Z    +0.000, E1   -76.269, E3 +16346.924}
SPL {X  -157.184, Y  +715.968, Z    +0.000, E1   -76.600, E3 +16442.882}
SPL {X  -156.461, Y  +718.560, Z    +0.000, E1   -75.553, E3 +16456.301}
SPL {X  -151.911, Y  +732.096, Z    +0.000, E1   -75.235, E3 +16466.856}
SPL {X  -146.569, Y  +744.407, Z    +0.000, E1   -74.677, E3 +16478.660}
SPL {X  -142.375, Y  +752.491, Z    +0.000, E1   -74.335, E3 +16485.687}
SPL {X  -139.539, Y  +757.399, Z    +0.000, E1   -73.892, E3 +16491.885}
SPL {X  -136.017, Y  +762.997, Z    +0.000, E1   -73.579, E3 +16497.067}
SPL {X  -133.089, Y  +767.296, Z    +0.000, E1   -73.251, E3 +16501.525}
SPL {X  -129.985, Y  +771.553, Z    +0.000, E1   -72.801, E3 +16506.519}
SPL {X  -126.581, Y  +775.909, Z    +0.000, E1   -72.426, E3 +16510.830}
SPL {X  -123.329, Y  +779.803, Z    +0.000, E1   -71.936, E3 +16515.212}
SPL {X  -119.291, Y  +784.315, Z    +0.000, E1   -72.148, E3 +16516.624}
SPL {X   -57.587, Y  +825.796, Z    +0.000, E1   -56.753, E3 +16670.386}
ENDSPLINE

SPLINE
SPL {X  -124.075, Y  +778.932, Z    +0.000, E1   -61.393, E3 +16864.015}
SPL {X  -150.653, Y  +735.257, Z    +0.000, E1   -50.160, E3 +16871.695}
SPL {X  -159.377, Y  +706.804, Z    +0.000, E1   -34.828, E3 +16873.338}
SPL {X  -162.134, Y  +688.425, Z    +0.000, E1   -19.100, E3 +16873.275}
SPL {X  -162.803, Y  +675.871, Z    +0.000, E1    -5.469, E3 +16873.459}
SPL {X  -162.820, Y  +671.500, Z    +0.000, E1    +0.000, E3 +16873.027}
SPL {X  -162.820, Y  +669.743, Z    +0.000, E1    +4.352, E3 +16872.822}
SPL {X  -162.820, Y  +665.917, Z    +0.000, E1   +15.272, E3 +16872.817}
SPL {X  -162.820, Y  +661.245, Z    +0.000, E1   +28.879, E3 +16872.658}
SPL {X  -162.820, Y  +654.015, Z    +0.000, E1   +45.814, E3 +16872.805}
SPL {X  -162.820, Y  +641.345, Z    +0.000, E1   +63.138, E3 +16872.852}
SPL {X  -162.820, Y  +620.039, Z    +0.000, E1   +75.979, E3 +16871.462}
SPL {X  -162.820, Y  +571.094, Z    +0.000, E1   +77.089, E3 +16886.641}
SPL {X  -157.487, Y  +339.169, Z    +0.000, E1   +76.425, E3 +16979.745}
SPL {X  -156.386, Y  +335.181, Z    +0.000, E1   +75.555, E3 +16991.805}
SPL {X  -152.710, Y  +324.020, Z    +0.000, E1   +75.365, E3 +16999.616}
SPL {X  -139.497, Y  +296.529, Z    +0.000, E1   +77.231, E3 +16993.188}
ENDSPLINE

SPLINE
SPL {X  -139.792, Y  +297.022, Z    +0.000, E1   +76.273, E3 +17001.883}
ENDSPLINE

SPLINE
SPL {X  -138.933, Y  +295.600, Z    +0.000, E1   +75.173, E3 +17012.365}
SPL {X  -137.186, Y  +292.805, Z    +0.000, E1   +73.993, E3 +17022.956}
SPL {X  -133.270, Y  +286.961, Z    +0.000, E1   +73.739, E3 +17027.669}
SPL {X  -130.283, Y  +282.844, Z    +0.000, E1   +73.297, E3 +17032.561}
SPL {X  -127.795, Y  +279.610, Z    +0.000, E1   +72.860, E3 +17036.691}
SPL {X  -124.650, Y  +275.749, Z    +0.000, E1   +72.674, E3 +17039.610}
SPL {X  -121.687, Y  +272.322, Z    +0.000, E1   +72.100, E3 +17043.919}
SPL {X  -113.980, Y  +264.229, Z    +0.000, E1   +74.120, E3 +17040.057}
SPL {X   -56.216, Y  +227.692, Z    +0.000, E1   +56.267, E3 +17216.781}
ENDSPLINE

SPLINE
SPL {X  -126.995, Y  +278.604, Z    +0.000, E1   +59.937, E3 +17389.021}
SPL {X  -150.196, Y  +317.640, Z    +0.000, E1   +49.956, E3 +17397.477}
SPL {X  -157.261, Y  +338.316, Z    +0.000, E1   +40.017, E3 +17399.172}
SPL {X  -160.924, Y  +355.726, Z    +0.000, E1   +27.715, E3 +17399.612}
SPL {X  -162.423, Y  +369.141, Z    +0.000, E1   +15.207, E3 +17400.048}
SPL {X  -162.811, Y  +378.755, Z    +0.000, E1    +4.616, E3 +17399.962}
SPL {X  -162.820, Y  +382.684, Z    +0.000, E1    -0.227, E3 +17399.517}
SPL {X  -162.820, Y  +387.227, Z    +0.000, E1   -12.320, E3 +17399.272}
SPL {X  -162.820, Y  +392.558, Z    +0.000, E1   -27.778, E3 +17399.308}
SPL {X  -162.820, Y  +400.474, Z    +0.000, E1   -46.251, E3 +17399.172}
SPL {X  -162.820, Y  +414.510, Z    +0.000, E1   -65.115, E3 +17398.615}
SPL {X  -162.820, Y  +465.064, Z    +0.000, E1   -76.269, E3 +17408.463}
SPL {X  -157.184, Y  +715.968, Z    +0.000, E1   -76.600, E3 +17504.420}
SPL {X  -156.461, Y  +718.560, Z    +0.000, E1   -75.553, E3 +17517.840}
SPL {X  -151.911, Y  +732.096, Z    +0.000, E1   -75.235, E3 +17528.394}
SPL {X  -146.569, Y  +744.407, Z    +0.000, E1   -74.677, E3 +17540.198}
SPL {X  -142.375, Y  +752.491, Z    +0.000, E1   -74.335, E3 +17547.226}
SPL {X  -139.539, Y  +757.399, Z    +0.000, E1   -73.892, E3 +17553.423}
SPL {X  -136.017, Y  +762.997, Z    +0.000, E1   -73.579, E3 +17558.606}
SPL {X  -133.089, Y  +767.296, Z    +0.000, E1   -73.251, E3 +17563.064}
SPL {X  -129.985, Y  +771.553, Z    +0.000, E1   -72.801, E3 +17568.057}
SPL {X  -126.581, Y  +775.909, Z    +0.000, E1   -72.426, E3 +17572.369}
SPL {X  -123.329, Y  +779.803, Z    +0.000, E1   -71.936, E3 +17576.750}
SPL {X  -119.291, Y  +784.315, Z    +0.000, E1   -72.148, E3 +17578.162}
SPL {X   -57.587, Y  +825.796, Z    +0.000, E1   -56.753, E3 +17731.925}
ENDSPLINE

SPLINE
SPL {X  -124.075, Y  +778.932, Z    +0.000, E1   -61.393, E3 +17925.554}
SPL {X  -150.653, Y  +735.257, Z    +0.000, E1   -50.160, E3 +17933.233}
SPL {X  -159.377, Y  +706.804, Z    +0.000, E1   -34.828, E3 +17934.876}
SPL {X  -162.134, Y  +688.425, Z    +0.000, E1   -19.100, E3 +17934.813}
SPL {X  -162.803, Y  +675.871, Z    +0.000, E1    -5.469, E3 +17934.997}
SPL {X  -162.820, Y  +671.500, Z    +0.000, E1    +0.000, E3 +17934.565}
SPL {X  -162.820, Y  +669.743, Z    +0.000, E1    +4.352, E3 +17934.361}
SPL {X  -162.820, Y  +665.917, Z    +0.000, E1   +15.272, E3 +17934.355}
SPL {X  -162.820, Y  +661.245, Z    +0.000, E1   +28.879, E3 +17934.197}
SPL {X  -162.820, Y  +654.015, Z    +0.000, E1   +45.814, E3 +17934.344}
SPL {X  -162.820, Y  +641.345, Z    +0.000, E1   +63.138, E3 +17934.391}
SPL {X  -162.820, Y  +620.039, Z    +0.000, E1   +75.979, E3 +17933.001}
SPL {X  -162.820, Y  +571.094, Z    +0.000, E1   +77.089, E3 +17948.179}
SPL {X  -157.487, Y  +339.169, Z    +0.000, E1   +76.425, E3 +18041.283}
SPL {X  -156.386, Y  +335.181, Z    +0.000, E1   +75.555, E3 +18053.344}
SPL {X  -152.710, Y  +324.020, Z    +0.000, E1   +75.365, E3 +18061.154}
SPL {X  -139.497, Y  +296.529, Z    +0.000, E1   +77.231, E3 +18054.726}
ENDSPLINE

SPLINE
SPL {X  -139.792, Y  +297.022, Z    +0.000, E1   +76.273, E3 +18063.421}
ENDSPLINE

SPLINE
SPL {X  -138.933, Y  +295.600, Z    +0.000, E1   +75.173, E3 +18073.904}
SPL {X  -137.186, Y  +292.805, Z    +0.000, E1   +73.993, E3 +18084.494}
SPL {X  -133.270, Y  +286.961, Z    +0.000, E1   +73.739, E3 +18089.208}
SPL {X  -130.283, Y  +282.844, Z    +0.000, E1   +73.297, E3 +18094.100}
SPL {X  -127.795, Y  +279.610, Z    +0.000, E1   +72.860, E3 +18098.230}
SPL {X  -124.650, Y  +275.749, Z    +0.000, E1   +72.674, E3 +18101.148}
SPL {X  -121.687, Y  +272.322, Z    +0.000, E1   +72.100, E3 +18105.457}
SPL {X  -113.980, Y  +264.229, Z    +0.000, E1   +74.120, E3 +18101.596}
SPL {X   -56.216, Y  +227.692, Z    +0.000, E1   +56.267, E3 +18278.320}
ENDSPLINE

SPLINE
SPL {X  -126.995, Y  +278.604, Z    +0.000, E1   +59.937, E3 +18450.560}
SPL {X  -150.196, Y  +317.640, Z    +0.000, E1   +49.956, E3 +18459.015}
SPL {X  -157.261, Y  +338.316, Z    +0.000, E1   +40.017, E3 +18460.710}
SPL {X  -160.924, Y  +355.726, Z    +0.000, E1   +27.715, E3 +18461.151}
SPL {X  -162.423, Y  +369.141, Z    +0.000, E1   +15.207, E3 +18461.586}
SPL {X  -162.811, Y  +378.755, Z    +0.000, E1    +4.616, E3 +18461.501}
SPL {X  -162.820, Y  +382.684, Z    +0.000, E1    -0.227, E3 +18461.055}
SPL {X  -162.820, Y  +387.227, Z    +0.000, E1   -12.320, E3 +18460.810}
SPL {X  -162.820, Y  +392.558, Z    +0.000, E1   -27.778, E3 +18460.846}
SPL {X  -162.820, Y  +400.474, Z    +0.000, E1   -46.251, E3 +18460.710}
SPL {X  -162.820, Y  +414.510, Z    +0.000, E1   -65.115, E3 +18460.153}
SPL {X  -162.820, Y  +465.064, Z    +0.000, E1   -76.269, E3 +18470.001}
SPL {X  -157.184, Y  +715.968, Z    +0.000, E1   -76.600, E3 +18565.959}
SPL {X  -156.461, Y  +718.560, Z    +0.000, E1   -75.553, E3 +18579.378}
SPL {X  -153.015, Y  +729.150, Z    +0.000, E1   -75.312, E3 +18587.468}
SPL {X  -149.053, Y  +739.025, Z    +0.000, E1   -74.952, E3 +18596.263}
SPL {X  -144.053, Y  +749.389, Z    +0.000, E1   -74.457, E3 +18606.255}
SPL {X  -139.539, Y  +757.399, Z    +0.000, E1   -73.892, E3 +18614.962}
SPL {X  -136.017, Y  +762.997, Z    +0.000, E1   -73.579, E3 +18620.144}
SPL {X  -133.089, Y  +767.296, Z    +0.000, E1   -73.251, E3 +18624.602}
SPL {X  -129.985, Y  +771.553, Z    +0.000, E1   -72.801, E3 +18629.596}
SPL {X  -126.581, Y  +775.909, Z    +0.000, E1   -72.426, E3 +18633.907}
SPL {X  -122.528, Y  +780.725, Z    +0.000, E1   -71.905, E3 +18638.927}
SPL {X  -116.189, Y  +787.563, Z    +0.000, E1   -72.978, E3 +18638.211}
SPL {X   -59.356, Y  +825.116, Z    +0.000, E1   -57.613, E3 +18774.356}
SPL {X   -56.547, Y  +826.185, Z    +0.000, E1   -55.989, E3 +18840.906}
ENDSPLINE

SPLINE
SPL {X  -124.075, Y  +778.932, Z    +0.000, E1   -61.393, E3 +18987.092}
SPL {X  -150.653, Y  +735.257, Z    +0.000, E1   -50.160, E3 +18994.772}
SPL {X  -159.377, Y  +706.804, Z    +0.000, E1   -34.828, E3 +18996.415}
SPL {X  -162.134, Y  +688.425, Z    +0.000, E1   -19.100, E3 +18996.352}
SPL {X  -162.734, Y  +678.779, Z    +0.000, E1    -8.745, E3 +18996.491}
SPL {X  -162.820, Y  +671.589, Z    +0.000, E1    -0.221, E3 +18996.125}
SPL {X  -162.820, Y  +669.743, Z    +0.000, E1    +4.352, E3 +18995.899}
SPL {X  -162.820, Y  +665.917, Z    +0.000, E1   +15.272, E3 +18995.894}
SPL {X  -162.820, Y  +659.880, Z    +0.000, E1   +32.256, E3 +18995.805}
SPL {X  -162.820, Y  +652.069, Z    +0.000, E1   +49.663, E3 +18995.831}
SPL {X  -162.820, Y  +641.345, Z    +0.000, E1   +63.138, E3 +18995.929}
SPL {X  -162.820, Y  +620.039, Z    +0.000, E1   +75.979, E3 +18994.539}
SPL {X  -162.820, Y  +578.479, Z    +0.000, E1   +77.260, E3 +19006.810}
SPL {X  -162.820, Y  +557.052, Z    +0.000, E1   +76.772, E3 +19015.291}
SPL {X  -157.487, Y  +339.169, Z    +0.000, E1   +76.425, E3 +19102.822}
SPL {X  -156.386, Y  +335.181, Z    +0.000, E1   +75.555, E3 +19114.882}
SPL {X  -152.710, Y  +324.020, Z    +0.000, E1   +75.365, E3 +19122.693}
SPL {X  -139.497, Y  +296.529, Z    +0.000, E1   +77.231, E3 +19116.264}
ENDSPLINE

SPLINE
SPL {X  -139.792, Y  +297.022, Z    +0.000, E1   +76.273, E3 +19124.960}
ENDSPLINE

SPLINE
SPL {X  -138.933, Y  +295.600, Z    +0.000, E1   +75.173, E3 +19135.442}
SPL {X  -137.186, Y  +292.805, Z    +0.000, E1   +73.993, E3 +19146.033}
SPL {X  -133.270, Y  +286.961, Z    +0.000, E1   +73.739, E3 +19150.746}
SPL {X  -130.283, Y  +282.844, Z    +0.000, E1   +73.297, E3 +19155.638}
SPL {X  -127.795, Y  +279.610, Z    +0.000, E1   +72.860, E3 +19159.768}
SPL {X  -124.650, Y  +275.749, Z    +0.000, E1   +72.674, E3 +19162.687}
SPL {X  -121.687, Y  +272.322, Z    +0.000, E1   +72.100, E3 +19166.996}
SPL {X  -113.980, Y  +264.229, Z    +0.000, E1   +74.120, E3 +19163.134}
SPL {X   -56.216, Y  +227.692, Z    +0.000, E1   +56.267, E3 +19339.858}
ENDSPLINE

SPLINE
SPL {X  -126.995, Y  +278.604, Z    +0.000, E1   +59.937, E3 +19512.098}
SPL {X  -150.196, Y  +317.640, Z    +0.000, E1   +49.956, E3 +19520.553}
SPL {X  -157.261, Y  +338.316, Z    +0.000, E1   +40.017, E3 +19522.249}
SPL {X  -160.924, Y  +355.726, Z    +0.000, E1   +27.715, E3 +19522.689}
SPL {X  -162.423, Y  +369.141, Z    +0.000, E1   +15.207, E3 +19523.125}
SPL {X  -162.811, Y  +378.755, Z    +0.000, E1    +4.616, E3 +19523.039}
SPL {X  -162.820, Y  +382.684, Z    +0.000, E1    -0.227, E3 +19522.594}
SPL {X  -162.820, Y  +385.721, Z    +0.000, E1    -8.371, E3 +19522.409}
SPL {X  -162.820, Y  +388.532, Z    +0.000, E1   -16.412, E3 +19522.296}
SPL {X  -162.820, Y  +392.558, Z    +0.000, E1   -27.778, E3 +19522.385}
SPL {X  -162.820, Y  +398.468, Z    +0.000, E1   -42.446, E3 +19522.235}
SPL {X  -162.820, Y  +404.415, Z    +0.000, E1   -53.236, E3 +19522.274}
SPL {X  -162.820, Y  +414.510, Z    +0.000, E1   -65.115, E3 +19521.692}
SPL {X  -162.820, Y  +457.766, Z    +0.000, E1   -75.929, E3 +19529.528}
SPL {X  -162.820, Y  +471.144, Z    +0.000, E1   -76.496, E3 +19533.217}
SPL {X  -158.097, Y  +712.432, Z    +0.000, E1   -77.677, E3 +19613.927}
SPL {X  -156.557, Y  +718.224, Z    +0.000, E1   -75.715, E3 +19639.064}
SPL {X  -153.015, Y  +729.150, Z    +0.000, E1   -75.312, E3 +19649.006}
SPL {X  -149.053, Y  +739.025, Z    +0.000, E1   -74.952, E3 +19657.802}
SPL {X  -145.525, Y  +746.527, Z    +0.000, E1   -74.526, E3 +19665.595}
SPL {X  -142.375, Y  +752.491, Z    +0.000, E1   -74.335, E3 +19670.303}
SPL {X  -139.539, Y  +757.399, Z    +0.000, E1   -73.892, E3 +19676.500}
SPL {X  -136.017, Y  +762.997, Z    +0.000, E1   -73.579, E3 +19681.683}
SPL {X  -133.089, Y  +767.296, Z    +0.000, E1   -73.251, E3 +19686.141}
SPL {X  -129.985, Y  +771.553, Z    +0.000, E1   -72.801, E3 +19691.134}
SPL {X  -126.581, Y  +775.909, Z    +0.000, E1   -72.426, E3 +19695.446}
SPL {X  -122.528, Y  +780.725, Z    +0.000, E1   -71.905, E3 +19700.466}
SPL {X  -116.189, Y  +787.563, Z    +0.000, E1   -72.978, E3 +19699.750}
SPL {X   -59.356, Y  +825.116, Z    +0.000, E1   -57.613, E3 +19835.895}
SPL {X   -56.547, Y  +826.185, Z    +0.000, E1   -55.989, E3 +19902.445}
ENDSPLINE

SPLINE
SPL {X  -124.075, Y  +778.932, Z    +0.000, E1   -61.393, E3 +20048.631}
SPL {X  -150.653, Y  +735.257, Z    +0.000, E1   -50.160, E3 +20056.310}
SPL {X  -159.377, Y  +706.804, Z    +0.000, E1   -34.828, E3 +20057.953}
SPL {X  -162.134, Y  +688.425, Z    +0.000, E1   -19.100, E3 +20057.890}
SPL {X  -162.734, Y  +678.779, Z    +0.000, E1    -8.745, E3 +20058.029}
SPL {X  -162.820, Y  +671.589, Z    +0.000, E1    -0.221, E3 +20057.664}
SPL {X  -162.820, Y  +669.743, Z    +0.000, E1    +4.352, E3 +20057.438}
SPL {X  -162.820, Y  +665.917, Z    +0.000, E1   +15.272, E3 +20057.432}
SPL {X  -162.820, Y  +659.880, Z    +0.000, E1   +32.256, E3 +20057.344}
SPL {X  -162.820, Y  +652.069, Z    +0.000, E1   +49.663, E3 +20057.369}
SPL {X  -162.820, Y  +641.345, Z    +0.000, E1   +63.138, E3 +20057.468}
SPL {X  -162.820, Y  +620.039, Z    +0.000, E1   +75.979, E3 +20056.078}
SPL {X  -162.820, Y  +571.094, Z    +0.000, E1   +77.089, E3 +20071.256}
SPL {X  -157.487, Y  +339.169, Z    +0.000, E1   +76.425, E3 +20164.360}
SPL {X  -156.386, Y  +335.181, Z    +0.000, E1   +75.555, E3 +20176.421}
SPL {X  -152.710, Y  +324.020, Z    +0.000, E1   +75.365, E3 +20184.231}
SPL {X  -139.497, Y  +296.529, Z    +0.000, E1   +77.231, E3 +20177.803}
ENDSPLINE

SPLINE
SPL {X  -139.520, Y  +296.568, Z    +0.000, E1   +75.884, E3 +20190.450}
ENDSPLINE

SPLINE
SPL {X  -138.554, Y  +294.984, Z    +0.000, E1   +74.772, E3 +20200.331}
SPL {X  -137.186, Y  +292.805, Z    +0.000, E1   +73.993, E3 +20207.571}
SPL {X  -133.270, Y  +286.961, Z    +0.000, E1   +73.739, E3 +20212.285}
SPL {X  -129.057, Y  +281.230, Z    +0.000, E1   +73.118, E3 +20219.192}
SPL {X  -123.859, Y  +274.815, Z    +0.000, E1   +72.511, E3 +20225.577}
SPL {X  -121.018, Y  +271.573, Z    +0.000, E1   +72.049, E3 +20229.094}
SPL {X  -113.980, Y  +264.229, Z    +0.000, E1   +74.120, E3 +20224.673}
SPL {X   -56.216, Y  +227.692, Z    +0.000, E1   +56.267, E3 +20401.397}
ENDSPLINE

SPLINE
SPL {X  -126.995, Y  +278.604, Z    +0.000, E1   +59.937, E3 +20573.637}
SPL {X  -150.196, Y  +317.640, Z    +0.000, E1   +49.956, E3 +20582.092}
SPL {X  -157.261, Y  +338.316, Z    +0.000, E1   +40.017, E3 +20583.787}
SPL {X  -160.924, Y  +355.726, Z    +0.000, E1   +27.715, E3 +20584.228}
SPL {X  -162.423, Y  +369.141, Z    +0.000, E1   +15.207, E3 +20584.663}
SPL {X  -162.811, Y  +378.755, Z    +0.000, E1    +4.616, E3 +20584.578}
SPL {X  -162.820, Y  +382.684, Z    +0.000, E1    -0.227, E3 +20584.132}
SPL {X  -162.820, Y  +387.227, Z    +0.000, E1   -12.320, E3 +20583.887}
SPL {X  -162.820, Y  +392.558, Z    +0.000, E1   -27.778, E3 +20583.923}
SPL {X  -162.820, Y  +400.474, Z    +0.000, E1   -46.251, E3 +20583.787}
SPL {X  -162.820, Y  +414.510, Z    +0.000, E1   -65.115, E3 +20583.230}
SPL {X  -162.820, Y  +465.064, Z    +0.000, E1   -76.269, E3 +20593.078}
SPL {X  -157.184, Y  +715.968, Z    +0.000, E1   -76.600, E3 +20689.036}
SPL {X  -156.461, Y  +718.560, Z    +0.000, E1   -75.553, E3 +20702.455}
SPL {X  -153.015, Y  +729.150, Z    +0.000, E1   -75.312, E3 +20710.544}
SPL {X  -149.053, Y  +739.025, Z    +0.000, E1   -74.952, E3 +20719.340}
SPL {X  -145.525, Y  +746.527, Z    +0.000, E1   -74.526, E3 +20727.134}
SPL {X  -142.375, Y  +752.491, Z    +0.000, E1   -74.335, E3 +20731.841}
SPL {X  -139.539, Y  +757.399, Z    +0.000, E1   -73.892, E3 +20738.039}
SPL {X  -136.017, Y  +762.997, Z    +0.000, E1   -73.579, E3 +20743.221}
SPL {X  -133.089, Y  +767.296, Z    +0.000, E1   -73.251, E3 +20747.679}
SPL {X  -129.985, Y  +771.553, Z    +0.000, E1   -72.801, E3 +20752.673}
SPL {X  -126.581, Y  +775.909, Z    +0.000, E1   -72.426, E3 +20756.984}
SPL {X  -122.528, Y  +780.725, Z    +0.000, E1   -71.905, E3 +20762.004}
SPL {X  -116.189, Y  +787.563, Z    +0.000, E1   -72.978, E3 +20761.288}
SPL {X   -59.356, Y  +825.116, Z    +0.000, E1   -57.613, E3 +20897.433}
SPL {X   -56.547, Y  +826.185, Z    +0.000, E1   -55.989, E3 +20963.983}
ENDSPLINE

SPLINE
SPL {X  -124.075, Y  +778.932, Z    +0.000, E1   -61.393, E3 +21110.169}
SPL {X  -150.653, Y  +735.257, Z    +0.000, E1   -50.160, E3 +21117.848}
SPL {X  -159.377, Y  +706.804, Z    +0.000, E1   -34.828, E3 +21119.492}
SPL {X  -162.134, Y  +688.425, Z    +0.000, E1   -19.100, E3 +21119.429}
SPL {X  -162.803, Y  +675.871, Z    +0.000, E1    -5.469, E3 +21119.613}
SPL {X  -162.820, Y  +671.500, Z    +0.000, E1    +0.000, E3 +21119.181}
SPL {X  -162.820, Y  +669.743, Z    +0.000, E1    +4.352, E3 +21118.976}
SPL {X  -162.820, Y  +665.917, Z    +0.000, E1   +15.272, E3 +21118.971}
SPL {X  -162.820, Y  +661.245, Z    +0.000, E1   +28.879, E3 +21118.812}
SPL {X  -162.820, Y  +654.015, Z    +0.000, E1   +45.814, E3 +21118.959}
SPL {X  -162.820, Y  +641.345, Z    +0.000, E1   +63.138, E3 +21119.006}
SPL {X  -162.820, Y  +620.039, Z    +0.000, E1   +75.979, E3 +21117.616}
SPL {X  -162.820, Y  +571.094, Z    +0.000, E1   +77.089, E3 +21132.795}
SPL {X  -157.487, Y  +339.169, Z    +0.000, E1   +76.425, E3 +21225.898}
SPL {X  -156.386, Y  +335.181, Z    +0.000, E1   +75.555, E3 +21237.959}
SPL {X  -152.710, Y  +324.020, Z    +0.000, E1   +75.365, E3 +21245.770}
SPL {X  -139.497, Y  +296.529, Z    +0.000, E1   +77.231, E3 +21239.341}
ENDSPLINE

SPLINE
SPL {X  -139.792, Y  +297.022, Z    +0.000, E1   +76.273, E3 +21248.037}
ENDSPLINE

SPLINE
SPL {X  -138.933, Y  +295.600, Z    +0.000, E1   +75.173, E3 +21258.519}
SPL {X  -137.186, Y  +292.805, Z    +0.000, E1   +73.993, E3 +21269.110}
SPL {X  -133.270, Y  +286.961, Z    +0.000, E1   +73.739, E3 +21273.823}
SPL {X  -130.283, Y  +282.844, Z    +0.000, E1   +73.297, E3 +21278.715}
SPL {X  -127.795, Y  +279.610, Z    +0.000, E1   +72.860, E3 +21282.845}
SPL {X  -124.650, Y  +275.749, Z    +0.000, E1   +72.674, E3 +21285.764}
SPL {X  -121.687, Y  +272.322, Z    +0.000, E1   +72.100, E3 +21290.073}
SPL {X  -113.980, Y  +264.229, Z    +0.000, E1   +74.120, E3 +21286.211}
SPL {X   -56.216, Y  +227.692, Z    +0.000, E1   +56.267, E3 +21462.935}
ENDSPLINE

SPLINE
SPL {X  -126.995, Y  +278.604, Z    +0.000, E1   +59.937, E3 +21635.175}
SPL {X  -150.196, Y  +317.640, Z    +0.000, E1   +49.956, E3 +21643.630}
SPL {X  -157.261, Y  +338.316, Z    +0.000, E1   +40.017, E3 +21645.326}
SPL {X  -160.924, Y  +355.726, Z    +0.000, E1   +27.715, E3 +21645.766}
SPL {X  -162.423, Y  +369.141, Z    +0.000, E1   +15.207, E3 +21646.202}
SPL {X  -162.811, Y  +378.755, Z    +0.000, E1    +4.616, E3 +21646.116}
SPL {X  -162.820, Y  +382.684, Z    +0.000, E1    -0.227, E3 +21645.671}
SPL {X  -162.820, Y  +387.227, Z    +0.000, E1   -12.320, E3 +21645.426}
SPL {X  -162.820, Y  +392.558, Z    +0.000, E1   -27.778, E3 +21645.462}
SPL {X  -162.820, Y  +400.474, Z    +0.000, E1   -46.251, E3 +21645.325}
SPL {X  -162.820, Y  +414.510, Z    +0.000, E1   -65.115, E3 +21644.769}
SPL {X  -162.820, Y  +465.064, Z    +0.000, E1   -76.269, E3 +21654.617}
SPL {X  -157.184, Y  +715.968, Z    +0.000, E1   -76.600, E3 +21750.574}
SPL {X  -156.461, Y  +718.560, Z    +0.000, E1   -75.553, E3 +21763.994}
SPL {X  -153.015, Y  +729.150, Z    +0.000, E1   -75.312, E3 +21772.083}
SPL {X  -149.053, Y  +739.025, Z    +0.000, E1   -74.952, E3 +21780.879}
SPL {X  -145.525, Y  +746.527, Z    +0.000, E1   -74.526, E3 +21788.672}
SPL {X  -142.375, Y  +752.491, Z    +0.000, E1   -74.335, E3 +21793.379}
SPL {X  -139.539, Y  +757.399, Z    +0.000, E1   -73.892, E3 +21799.577}
SPL {X  -136.017, Y  +762.997, Z    +0.000, E1   -73.579, E3 +21804.759}
SPL {X  -133.089, Y  +767.296, Z    +0.000, E1   -73.251, E3 +21809.218}
SPL {X  -129.985, Y  +771.553, Z    +0.000, E1   -72.801, E3 +21814.211}
SPL {X  -126.581, Y  +775.909, Z    +0.000, E1   -72.426, E3 +21818.522}
SPL {X  -123.329, Y  +779.803, Z    +0.000, E1   -71.936, E3 +21822.904}
SPL {X  -119.291, Y  +784.315, Z    +0.000, E1   -72.148, E3 +21824.316}
SPL {X   -57.587, Y  +825.796, Z    +0.000, E1   -56.753, E3 +21978.079}
ENDSPLINE

SPLINE
SPL {X  -124.075, Y  +778.932, Z    +0.000, E1   -61.393, E3 +22171.708}
SPL {X  -150.653, Y  +735.257, Z    +0.000, E1   -50.160, E3 +22179.387}
SPL {X  -159.377, Y  +706.804, Z    +0.000, E1   -34.828, E3 +22181.030}
SPL {X  -162.134, Y  +688.425, Z    +0.000, E1   -19.100, E3 +22180.967}
SPL {X  -162.803, Y  +675.871, Z    +0.000, E1    -5.469, E3 +22181.151}
SPL {X  -162.820, Y  +671.500, Z    +0.000, E1    +0.000, E3 +22180.719}
SPL {X  -162.820, Y  +669.743, Z    +0.000, E1    +4.352, E3 +22180.515}
SPL {X  -162.820, Y  +665.917, Z    +0.000, E1   +15.272, E3 +22180.509}
SPL {X  -162.820, Y  +661.245, Z    +0.000, E1   +28.879, E3 +22180.350}
SPL {X  -162.820, Y  +654.015, Z    +0.000, E1   +45.814, E3 +22180.498}
SPL {X  -162.820, Y  +641.345, Z    +0.000, E1   +63.138, E3 +22180.545}
SPL {X  -162.820, Y  +620.039, Z    +0.000, E1   +75.979, E3 +22179.154}
SPL {X  -162.820, Y  +578.479, Z    +0.000, E1   +77.260, E3 +22191.425}
SPL {X  -162.820, Y  +557.052, Z    +0.000, E1   +76.772, E3 +22199.906}
SPL {X  -157.487, Y  +339.169, Z    +0.000, E1   +76.425, E3 +22287.437}
SPL {X  -156.386, Y  +335.181, Z    +0.000, E1   +75.555, E3 +22299.498}
SPL {X  -152.710, Y  +324.020, Z    +0.000, E1   +75.365, E3 +22307.308}
SPL {X  -139.497, Y  +296.529, Z    +0.000, E1   +77.231, E3 +22300.880}
ENDSPLINE

SPLINE
SPL {X  -139.792, Y  +297.022, Z    +0.000, E1   +76.273, E3 +22309.575}
ENDSPLINE

SPLINE
SPL {X  -138.933, Y  +295.600, Z    +0.000, E1   +75.173, E3 +22320.058}
SPL {X  -137.186, Y  +292.805, Z    +0.000, E1   +73.993, E3 +22330.648}
SPL {X  -133.270, Y  +286.961, Z    +0.000, E1   +73.739, E3 +22335.362}
SPL {X  -130.283, Y  +282.844, Z    +0.000, E1   +73.297, E3 +22340.253}
SPL {X  -126.880, Y  +278.461, Z    +0.000, E1   +72.855, E3 +22345.004}
SPL {X  -124.135, Y  +275.140, Z    +0.000, E1   +72.554, E3 +22348.132}
SPL {X  -121.687, Y  +272.322, Z    +0.000, E1   +72.100, E3 +22351.611}
SPL {X  -113.980, Y  +264.229, Z    +0.000, E1   +74.120, E3 +22347.750}
SPL {X   -56.216, Y  +227.692, Z    +0.000, E1   +56.267, E3 +22524.474}
ENDSPLINE

SPLINE
SPL {X  -126.995, Y  +278.604, Z    +0.000, E1   +59.937, E3 +22696.714}
SPL {X  -150.196, Y  +317.640, Z    +0.000, E1   +49.956, E3 +22705.169}
SPL {X  -157.261, Y  +338.316, Z    +0.000, E1   +40.017, E3 +22706.864}
SPL {X  -160.924, Y  +355.726, Z    +0.000, E1   +27.715, E3 +22707.305}
SPL {X  -162.423, Y  +369.141, Z    +0.000, E1   +15.207, E3 +22707.740}
SPL {X  -162.811, Y  +378.755, Z    +0.000, E1    +4.616, E3 +22707.655}
SPL {X  -162.820, Y  +382.684, Z    +0.000, E1    -0.227, E3 +22707.209}
SPL {X  -162.820, Y  +385.721, Z    +0.000, E1    -8.371, E3 +22707.025}
SPL {X  -162.820, Y  +388.532, Z    +0.000, E1   -16.412, E3 +22706.911}
SPL {X  -162.820, Y  +392.558, Z    +0.000, E1   -27.778, E3 +22707.000}
SPL {X  -162.820, Y  +400.474, Z    +0.000, E1   -46.251, E3 +22706.864}
SPL {X  -162.820, Y  +414.510, Z    +0.000, E1   -65.115, E3 +22706.307}
SPL {X  -162.820, Y  +465.064, Z    +0.000, E1   -76.269, E3 +22716.155}
SPL {X  -157.184, Y  +715.968, Z    +0.000, E1   -76.600, E3 +22812.112}
SPL {X  -156.461, Y  +718.560, Z    +0.000, E1   -75.553, E3 +22825.532}
SPL {X  -153.015, Y  +729.150, Z    +0.000, E1   -75.312, E3 +22833.621}
SPL {X  -149.053, Y  +739.025, Z    +0.000, E1   -74.952, E3 +22842.417}
SPL {X  -144.053, Y  +749.389, Z    +0.000, E1   -74.457, E3 +22852.409}
SPL {X  -139.539, Y  +757.399, Z    +0.000, E1   -73.892, E3 +22861.116}
SPL {X  -136.017, Y  +762.997, Z    +0.000, E1   -73.579, E3 +22866.298}
SPL {X  -133.089, Y  +767.296, Z    +0.000, E1   -73.251, E3 +22870.756}
SPL {X  -129.985, Y  +771.553, Z    +0.000, E1   -72.801, E3 +22875.750}
SPL {X  -126.581, Y  +775.909, Z    +0.000, E1   -72.426, E3 +22880.061}
SPL {X  -123.329, Y  +779.803, Z    +0.000, E1   -71.936, E3 +22884.443}
SPL {X  -119.291, Y  +784.315, Z    +0.000, E1   -72.148, E3 +22885.855}
SPL {X   -57.587, Y  +825.796, Z    +0.000, E1   -56.753, E3 +23039.617}
ENDSPLINE

SPLINE
SPL {X  -124.075, Y  +778.932, Z    +0.000, E1   -61.393, E3 +23233.246}
SPL {X  -147.028, Y  +743.450, Z    +0.000, E1   -53.078, E3 +23239.983}
SPL {X  -152.552, Y  +730.406, Z    +0.000, E1   -48.136, E3 +23241.401}
SPL {X  -159.377, Y  +706.804, Z    +0.000, E1   -34.828, E3 +23242.569}
SPL {X  -162.134, Y  +688.425, Z    +0.000, E1   -19.100, E3 +23242.506}
SPL {X  -162.803, Y  +675.871, Z    +0.000, E1    -5.469, E3 +23242.690}
SPL {X  -162.820, Y  +671.500, Z    +0.000, E1    +0.000, E3 +23242.258}
SPL {X  -162.820, Y  +669.743, Z    +0.000, E1    +4.352, E3 +23242.053}
SPL {X  -162.820, Y  +665.917, Z    +0.000, E1   +15.272, E3 +23242.048}
SPL {X  -162.820, Y  +661.245, Z    +0.000, E1   +28.879, E3 +23241.889}
SPL {X  -162.820, Y  +654.015, Z    +0.000, E1   +45.814, E3 +23242.036}
SPL {X  -162.820, Y  +641.345, Z    +0.000, E1   +63.138, E3 +23242.083}
SPL {X  -162.820, Y  +620.039, Z    +0.000, E1   +75.979, E3 +23240.693}
SPL {X  -162.820, Y  +571.094, Z    +0.000, E1   +77.089, E3 +23255.872}
SPL {X  -157.487, Y  +339.169, Z    +0.000, E1   +76.425, E3 +23348.975}
SPL {X  -156.386, Y  +335.181, Z    +0.000, E1   +75.555, E3 +23361.036}
SPL {X  -152.710, Y  +324.020, Z    +0.000, E1   +75.365, E3 +23368.847}
SPL {X  -139.497, Y  +296.529, Z    +0.000, E1   +77.231, E3 +23362.418}
ENDSPLINE

SPLINE
SPL {X  -139.792, Y  +297.022, Z    +0.000, E1   +76.273, E3 +23371.113}
ENDSPLINE

SPLINE
SPL {X  -138.933, Y  +295.600, Z    +0.000, E1   +75.173, E3 +23381.596}
SPL {X  -137.186, Y  +292.805, Z    +0.000, E1   +73.993, E3 +23392.187}
SPL {X  -133.270, Y  +286.961, Z    +0.000, E1   +73.739, E3 +23396.900}
SPL {X  -130.283, Y  +282.844, Z    +0.000, E1   +73.297, E3 +23401.792}
SPL {X  -126.880, Y  +278.461, Z    +0.000, E1   +72.855, E3 +23406.542}
SPL {X  -123.363, Y  +274.237, Z    +0.000, E1   +72.376, E3 +23411.024}
SPL {X  -121.018, Y  +271.573, Z    +0.000, E1   +72.049, E3 +23413.710}
SPL {X  -113.980, Y  +264.229, Z    +0.000, E1   +74.120, E3 +23409.288}
SPL {X   -56.216, Y  +227.692, Z    +0.000, E1   +56.267, E3 +23586.012}
ENDSPLINE

SPLINE
SPL {X  -126.995, Y  +278.604, Z    +0.000, E1   +59.937, E3 +23758.252}
SPL {X  -150.196, Y  +317.640, Z    +0.000, E1   +49.956, E3 +23766.707}
SPL {X  -157.261, Y  +338.316, Z    +0.000, E1   +40.017, E3 +23768.402}
SPL {X  -160.924, Y  +355.726, Z    +0.000, E1   +27.715, E3 +23768.843}
SPL {X  -162.423, Y  +369.141, Z    +0.000, E1   +15.207, E3 +23769.279}
SPL {X  -162.811, Y  +378.755, Z    +0.000, E1    +4.616, E3 +23769.193}
SPL {X  -162.820, Y  +382.684, Z    +0.000, E1    -0.227, E3 +23768.748}
SPL {X  -162.820, Y  +385.721, Z    +0.000, E1    -8.371, E3 +23768.563}
SPL {X  -162.820, Y  +388.532, Z    +0.000, E1   -16.412, E3 +23768.450}
SPL {X  -162.820, Y  +392.558, Z    +0.000, E1   -27.778, E3 +23768.539}
SPL {X  -162.820, Y  +400.474, Z    +0.000, E1   -46.251, E3 +23768.402}
SPL {X  -162.820, Y  +414.510, Z    +0.000, E1   -65.115, E3 +23767.845}
SPL {X  -162.820, Y  +465.064, Z    +0.000, E1   -76.269, E3 +23777.693}
SPL {X  -157.184, Y  +715.968, Z    +0.000, E1   -76.600, E3 +23873.651}
SPL {X  -156.461, Y  +718.560, Z    +0.000, E1   -75.553, E3 +23887.071}
SPL {X  -151.911, Y  +732.096, Z    +0.000, E1   -75.235, E3 +23897.625}
SPL {X  -146.569, Y  +744.407, Z    +0.000, E1   -74.677, E3 +23909.429}
SPL {X  -142.375, Y  +752.491, Z    +0.000, E1   -74.335, E3 +23916.456}
SPL {X  -139.539, Y  +757.399, Z    +0.000, E1   -73.892, E3 +23922.654}
SPL {X  -136.017, Y  +762.997, Z    +0.000, E1   -73.579, E3 +23927.836}
SPL {X  -133.089, Y  +767.296, Z    +0.000, E1   -73.251, E3 +23932.294}
SPL {X  -129.985, Y  +771.553, Z    +0.000, E1   -72.801, E3 +23937.288}
SPL {X  -126.581, Y  +775.909, Z    +0.000, E1   -72.426, E3 +23941.599}
SPL {X  -122.528, Y  +780.725, Z    +0.000, E1   -71.905, E3 +23946.619}
SPL {X  -116.189, Y  +787.563, Z    +0.000, E1   -72.978, E3 +23945.904}
SPL {X   -57.587, Y  +825.796, Z    +0.000, E1   -56.753, E3 +24101.156}
ENDSPLINE

SPLINE
SPL {X  -124.075, Y  +778.932, Z    +0.000, E1   -61.393, E3 +24294.785}
SPL {X  -147.028, Y  +743.450, Z    +0.000, E1   -53.078, E3 +24301.522}
SPL {X  -152.552, Y  +730.406, Z    +0.000, E1   -48.136, E3 +24302.939}
SPL {X  -159.377, Y  +706.804, Z    +0.000, E1   -34.828, E3 +24304.107}
SPL {X  -162.134, Y  +688.425, Z    +0.000, E1   -19.100, E3 +24304.044}
SPL {X  -162.803, Y  +675.871, Z    +0.000, E1    -5.469, E3 +24304.228}
SPL {X  -162.820, Y  +671.500, Z    +0.000, E1    +0.000, E3 +24303.796}
SPL {X  -162.820, Y  +669.743, Z    +0.000, E1    +4.352, E3 +24303.592}
SPL {X  -162.820, Y  +665.917, Z    +0.000, E1   +15.272, E3 +24303.586}
SPL {X  -162.820, Y  +661.245, Z    +0.000, E1   +28.879, E3 +24303.427}
SPL {X  -162.820, Y  +654.015, Z    +0.000, E1   +45.814, E3 +24303.574}
SPL {X  -162.820, Y  +641.345, Z    +0.000, E1   +63.138, E3 +24303.622}
SPL {X  -162.820, Y  +620.039, Z    +0.000, E1   +75.979, E3 +24302.231}
SPL {X  -162.820, Y  +571.094, Z    +0.000, E1   +77.089, E3 +24317.410}
SPL {X  -157.487, Y  +339.169, Z    +0.000, E1   +76.425, E3 +24410.514}
SPL {X  -156.386, Y  +335.181, Z    +0.000, E1   +75.555, E3 +24422.575}
SPL {X  -152.710, Y  +324.020, Z    +0.000, E1   +75.365, E3 +24430.385}
SPL {X  -139.497, Y  +296.529, Z    +0.000, E1   +77.231, E3 +24423.957}
ENDSPLINE

SPLINE
SPL {X  -139.520, Y  +296.568, Z    +0.000, E1   +75.884, E3 +24436.604}
ENDSPLINE

SPLINE
SPL {X  -138.554, Y  +294.984, Z    +0.000, E1   +74.772, E3 +24446.485}
SPL {X  -137.186, Y  +292.805, Z    +0.000, E1   +73.993, E3 +24453.725}
SPL {X  -133.270, Y  +286.961, Z    +0.000, E1   +73.739, E3 +24458.438}
SPL {X  -130.283, Y  +282.844, Z    +0.000, E1   +73.297, E3 +24463.330}
SPL {X  -127.795, Y  +279.610, Z    +0.000, E1   +72.860, E3 +24467.461}
SPL {X  -124.650, Y  +275.749, Z    +0.000, E1   +72.674, E3 +24470.379}
SPL {X  -121.687, Y  +272.322, Z    +0.000, E1   +72.100, E3 +24474.688}
SPL {X  -113.980, Y  +264.229, Z    +0.000, E1   +74.120, E3 +24470.826}
SPL {X   -56.216, Y  +227.692, Z    +0.000, E1   +56.267, E3 +24647.550}
ENDSPLINE

SPLINE
SPL {X  -126.995, Y  +278.604, Z    +0.000, E1   +59.937, E3 +24819.791}
SPL {X  -150.196, Y  +317.640, Z    +0.000, E1   +49.956, E3 +24828.246}
SPL {X  -157.261, Y  +338.316, Z    +0.000, E1   +40.017, E3 +24829.941}
SPL {X  -160.924, Y  +355.726, Z    +0.000, E1   +27.715, E3 +24830.382}
SPL {X  -162.423, Y  +369.141, Z    +0.000, E1   +15.207, E3 +24830.817}
SPL {X  -162.811, Y  +378.755, Z    +0.000, E1    +4.616, E3 +24830.732}
SPL {X  -162.820, Y  +382.684, Z    +0.000, E1    -0.227, E3 +24830.286}
SPL {X  -162.820, Y  +387.227, Z    +0.000, E1   -12.320, E3 +24830.041}
SPL {X  -162.820, Y  +392.558, Z    +0.000, E1   -27.778, E3 +24830.077}
SPL {X  -162.820, Y  +400.474, Z    +0.000, E1   -46.251, E3 +24829.941}
SPL {X  -162.820, Y  +414.510, Z    +0.000, E1   -65.115, E3 +24829.384}
SPL {X  -162.820, Y  +465.064, Z    +0.000, E1   -76.269, E3 +24839.232}
SPL {X  -157.184, Y  +715.968, Z    +0.000, E1   -76.600, E3 +24935.189}
SPL {X  -156.461, Y  +718.560, Z    +0.000, E1   -75.553, E3 +24948.609}
SPL {X  -151.911, Y  +732.096, Z    +0.000, E1   -75.235, E3 +24959.163}
SPL {X  -146.569, Y  +744.407, Z    +0.000, E1   -74.677, E3 +24970.967}
SPL {X  -142.375, Y  +752.491, Z    +0.000, E1   -74.335, E3 +24977.995}
SPL {X  -139.539, Y  +757.399, Z    +0.000, E1   -73.892, E3 +24984.192}
SPL {X  -136.017, Y  +762.997, Z    +0.000, E1   -73.579, E3 +24989.375}
SPL {X  -133.089, Y  +767.296, Z    +0.000, E1   -73.251, E3 +24993.833}
SPL {X  -129.985, Y  +771.553, Z    +0.000, E1   -72.801, E3 +24998.827}
SPL {X  -126.581, Y  +775.909, Z    +0.000, E1   -72.426, E3 +25003.138}
SPL {X  -122.528, Y  +780.725, Z    +0.000, E1   -71.905, E3 +25008.158}
SPL {X  -116.189, Y  +787.563, Z    +0.000, E1   -72.978, E3 +25007.442}
SPL {X   -59.356, Y  +825.116, Z    +0.000, E1   -57.613, E3 +25143.587}
SPL {X   -56.547, Y  +826.185, Z    +0.000, E1   -55.989, E3 +25210.137}
ENDSPLINE

SPLINE
SPL {X  -124.075, Y  +778.932, Z    +0.000, E1   -61.393, E3 +25356.323}
SPL {X  -150.653, Y  +735.257, Z    +0.000, E1   -50.160, E3 +25364.002}
SPL {X  -159.377, Y  +706.804, Z    +0.000, E1   -34.828, E3 +25365.646}
SPL {X  -162.134, Y  +688.425, Z    +0.000, E1   -19.100, E3 +25365.583}
SPL {X  -162.734, Y  +678.779, Z    +0.000, E1    -8.745, E3 +25365.722}
SPL {X  -162.820, Y  +671.589, Z    +0.000, E1    -0.221, E3 +25365.356}
SPL {X  -162.820, Y  +669.743, Z    +0.000, E1    +4.352, E3 +25365.130}
SPL {X  -162.820, Y  +665.917, Z    +0.000, E1   +15.272, E3 +25365.125}
SPL {X  -162.820, Y  +661.245, Z    +0.000, E1   +28.879, E3 +25364.966}
SPL {X  -162.820, Y  +654.015, Z    +0.000, E1   +45.814, E3 +25365.113}
SPL {X  -162.820, Y  +641.345, Z    +0.000, E1   +63.138, E3 +25365.160}
SPL {X  -162.820, Y  +620.039, Z    +0.000, E1   +75.979, E3 +25363.770}
SPL {X  -162.820, Y  +571.094, Z    +0.000, E1   +77.089, E3 +25378.948}
SPL {X  -157.487, Y  +339.169, Z    +0.000, E1   +76.425, E3 +25472.052}
SPL {X  -156.386, Y  +335.181, Z    +0.000, E1   +75.555, E3 +25484.113}
SPL {X  -152.710, Y  +324.020, Z    +0.000, E1   +75.365, E3 +25491.924}
SPL {X  -139.497, Y  +296.529, Z    +0.000, E1   +77.231, E3 +25485.495}
ENDSPLINE

SPLINE
SPL {X  -139.792, Y  +297.022, Z    +0.000, E1   +76.273, E3 +25494.190}
ENDSPLINE

SPLINE
SPL {X  -138.933, Y  +295.600, Z    +0.000, E1   +75.173, E3 +25504.673}
SPL {X  -137.186, Y  +292.805, Z    +0.000, E1   +73.993, E3 +25515.264}
SPL {X  -133.270, Y  +286.961, Z    +0.000, E1   +73.739, E3 +25519.977}
SPL {X  -130.283, Y  +282.844, Z    +0.000, E1   +73.297, E3 +25524.869}
SPL {X  -126.880, Y  +278.461, Z    +0.000, E1   +72.855, E3 +25529.619}
SPL {X  -123.363, Y  +274.237, Z    +0.000, E1   +72.376, E3 +25534.101}
SPL {X  -121.018, Y  +271.573, Z    +0.000, E1   +72.049, E3 +25536.787}
SPL {X  -113.980, Y  +264.229, Z    +0.000, E1   +74.120, E3 +25532.365}
SPL {X   -56.216, Y  +227.692, Z    +0.000, E1   +56.267, E3 +25709.089}
ENDSPLINE

SPLINE
SPL {X  -126.995, Y  +278.604, Z    +0.000, E1   +59.937, E3 +25881.329}
SPL {X  -150.196, Y  +317.640, Z    +0.000, E1   +49.956, E3 +25889.784}
SPL {X  -157.261, Y  +338.316, Z    +0.000, E1   +40.017, E3 +25891.479}
SPL {X  -160.924, Y  +355.726, Z    +0.000, E1   +27.715, E3 +25891.920}
SPL {X  -162.423, Y  +369.141, Z    +0.000, E1   +15.207, E3 +25892.356}
SPL {X  -162.811, Y  +378.755, Z    +0.000, E1    +4.616, E3 +25892.270}
SPL {X  -162.820, Y  +382.684, Z    +0.000, E1    -0.227, E3 +25891.825}
SPL {X  -162.820, Y  +387.227, Z    +0.000, E1   -12.320, E3 +25891.579}
SPL {X  -162.820, Y  +392.558, Z    +0.000, E1   -27.778, E3 +25891.616}
SPL {X  -162.820, Y  +400.474, Z    +0.000, E1   -46.251, E3 +25891.479}
SPL {X  -162.820, Y  +414.510, Z    +0.000, E1   -65.115, E3 +25890.922}
SPL {X  -162.820, Y  +465.064, Z    +0.000, E1   -76.269, E3 +25900.770}
SPL {X  -157.184, Y  +715.968, Z    +0.000, E1   -76.600, E3 +25996.728}
SPL {X  -156.461, Y  +718.560, Z    +0.000, E1   -75.553, E3 +26010.148}
SPL {X  -151.911, Y  +732.096, Z    +0.000, E1   -75.235, E3 +26020.702}
SPL {X  -146.569, Y  +744.407, Z    +0.000, E1   -74.677, E3 +26032.506}
SPL {X  -142.375, Y  +752.491, Z    +0.000, E1   -74.335, E3 +26039.533}
SPL {X  -139.539, Y  +757.399, Z    +0.000, E1   -73.892, E3 +26045.731}
SPL {X  -136.017, Y  +762.997, Z    +0.000, E1   -73.579, E3 +26050.913}
SPL {X  -133.089, Y  +767.296, Z    +0.000, E1   -73.251, E3 +26055.371}
SPL {X  -129.985, Y  +771.553, Z    +0.000, E1   -72.801, E3 +26060.365}
SPL {X  -126.581, Y  +775.909, Z    +0.000, E1   -72.426, E3 +26064.676}
SPL {X  -123.329, Y  +779.803, Z    +0.000, E1   -71.936, E3 +26069.058}
SPL {X  -119.291, Y  +784.315, Z    +0.000, E1   -72.148, E3 +26070.470}
SPL {X   -57.587, Y  +825.796, Z    +0.000, E1   -56.753, E3 +26224.233}
ENDSPLINE

